  MoveL 7815 to (31.1, 13.35, -12.25) mm, rotated rx -180 ry 0 rz 90 deg; joints [74.527, -16.728, 82.289, 0, 24.439, 74.527]
  MoveL 7816 to (23.55, 13.35, -12.25) mm, rotated rx 180 ry 0 rz 90 deg; joints [74.46, -16.875, 82.836, 0, 24.039, 74.46]
  MoveL 7817 to (23.55, 15.07, -12.25) mm, rotated rx -180 ry 0 rz 90 deg; joints [74.516, -16.884, 82.871, 0, 24.013, 74.516]
  MoveL 7818 to (23.55, 15.07, -9.25) mm, rotated rx 180 ry 0 rz 90 deg; joints [74.516, -17.037, 82.973, 0, 24.064, 74.516]
  Establecer velocidad (1000.0 mm/s)
  MoveL 7819 to (23.55, 15.07, 10) mm, rotated rx 180 ry 0 rz 90 deg; joints [74.516, -18.015, 83.619, 0, 24.396, 74.516]
  Establecer velocidad (66.7 mm/s)
  MoveL 7820 to (-7.83, 65.77, 10) mm, rotated rx -180 ry 0 rz 90 deg; joints [75.899, -18.849, 86.805, 0, 22.044, 75.899]
  MoveL 7821 to (-7.83, 65.77, -9) mm, rotated rx 180 ry 0 rz 90 deg; joints [75.899, -17.87, 86.169, 0, 21.701, 75.899]
  MoveL 7822 to (-8.11, 64.28, -9.41) mm, rotated rx -180 ry 0 rz 90 deg; joints [75.847, -17.848, 86.149, 0, 21.699, 75.847]
  MoveL 7823 to (-7.99, 62.77, -9.81) mm, rotated rx -180 ry 0 rz 90 deg; joints [75.798, -17.818, 86.1, 0, 21.718, 75.798]
  MoveL 7824 to (-7.51, 61.33, -10.22) mm, rotated rx 180 ry 0 rz 90 deg; joints [75.754, -17.782, 86.027, 0, 21.756, 75.754]
  MoveL 7825 to (-6.7, 60.05, -10.62) mm, rotated rx -180 ry 0 rz 90 deg; joints [75.719, -17.742, 85.933, 0, 21.809, 75.719]
  MoveL 7826 to (-5.59, 59, -11.03) mm, rotated rx 180 ry 0 rz 90 deg; joints [75.693, -17.697, 85.823, 0, 21.874, 75.693]
  MoveL 7827 to (-4.27, 58.25, -11.44) mm, rotated rx -180 ry 0 rz 90 deg; joints [75.68, -17.649, 85.702, 0, 21.947, 75.68]
  MoveL 7828 to (-2.8, 57.85, -11.84) mm, rotated rx 180 ry 0 rz 90 deg; joints [75.679, -17.601, 85.578, 0, 22.023, 75.679]
  MoveL 7829 to (-1.29, 57.84, -12.25) mm, rotated rx 180 ry 0 rz 90 deg; joints [75.691, -17.553, 85.457, 0, 22.096, 75.691]
  MoveL 7830 to (6.58, 58.62, -12.25) mm, rotated rx 180 ry 0 rz 90 deg; joints [75.783, -17.416, 84.913, 0, 22.503, 75.783]
  MoveC 7831 to (18.86, 59.96, -12.25) mm, rotated rx 180 ry 0 rz 90 deg; joints [75.928, -17.197, 84.061, 0, 23.136, 75.928] to (31.1, 61.55, -12.25) mm, rotated rx -180 ry 0 rz 90 deg; joints [76.079, -16.973, 83.207, 0, 23.766, 76.079]
  MoveL 7832 to (31.1, 68.78, -12.25) mm, rotated rx 180 ry 0 rz 90 deg; joints [76.313, -17.007, 83.336, 0, 23.672, 76.313]
  MoveC 7833 to (8.53, 69.82, -12.25) mm, rotated rx -180 ry 0 rz 90 deg; joints [76.167, -17.432, 84.974, 0, 22.457, 76.167] to (-14.06, 70.54, -12.25) mm, rotated rx -180 ry 0 rz 90 deg; joints [76.005, -17.83, 86.579, 0, 21.251, 76.005]
  MoveC 7834 to (-16.19, 67.95, -12.25) mm, rotated rx -180 ry 0 rz 90 deg; joints [75.901, -17.855, 86.682, 0, 21.173, 75.901] to (-15.95, 64.6, -12.25) mm, rotated rx 180 ry 0 rz 90 deg; joints [75.792, -17.836, 86.606, 0, 21.231, 75.792]
  MoveL 7835 to (-7.11, 58.83, -12.25) mm, rotated rx 180 ry 0 rz 90 deg; joints [75.675, -17.66, 85.884, 0, 21.775, 75.675]
  MoveL 7836 to (-5.82, 57.95, -12.25) mm, rotated rx -180 ry 0 rz 90 deg; joints [75.657, -17.633, 85.778, 0, 21.855, 75.657]
  MoveC 7837 to (-5.45, 57.71, -12.25) mm, rotated rx 180 ry 0 rz 90 deg; joints [75.652, -17.626, 85.747, 0, 21.878, 75.652] to (-5.05, 57.51, -12.25) mm, rotated rx -180 ry 0 rz 90 deg; joints [75.649, -17.618, 85.716, 0, 21.902, 75.649]
  MoveC 7838 to (0.56, 58.01, -12.25) mm, rotated rx 180 ry 0 rz 90 deg; joints [75.713, -17.521, 85.329, 0, 22.192, 75.713] to (6.16, 58.57, -12.25) mm, rotated rx -180 ry 0 rz 90 deg; joints [75.778, -17.424, 84.943, 0, 22.481, 75.778]
  MoveC 7839 to (6.37, 58.59, -12.25) mm, rotated rx 180 ry 0 rz 90 deg; joints [75.78, -17.42, 84.928, 0, 22.492, 75.78] to (6.58, 58.62, -12.25) mm, rotated rx 180 ry 0 rz 90 deg; joints [75.783, -17.416, 84.913, 0, 22.503, 75.783]
  MoveL 7840 to (5.83, 66.13, -12.25) mm, rotated rx -180 ry 0 rz 90 deg; joints [76.023, -17.464, 85.101, 0, 22.363, 76.023]
  MoveL 7841 to (5.83, 66.13, -9.25) mm, rotated rx 180 ry 0 rz 90 deg; joints [76.023, -17.618, 85.203, 0, 22.415, 76.023]
  Establecer velocidad (1000.0 mm/s)
  MoveL 7842 to (5.83, 66.13, 10) mm, rotated rx 180 ry 0 rz 90 deg; joints [76.023, -18.605, 85.848, 0, 22.757, 76.023]
  Establecer velocidad (66.7 mm/s)
  MoveL 7843 to (-63.61, 35.65, 10) mm, rotated rx 180 ry 0 rz 90 deg; joints [74.395, -19.637, 90.091, 0, 19.546, 74.395]
  MoveL 7844 to (-63.61, 35.65, -9) mm, rotated rx 180 ry 0 rz 90 deg; joints [74.395, -18.644, 89.455, 0, 19.189, 74.395]
  MoveL 7845 to (-65.12, 35.84, -9.41) mm, rotated rx -180 ry 0 rz 90 deg; joints [74.387, -18.646, 89.546, 0, 19.1, 74.387]
  MoveL 7846 to (-66.63, 35.66, -9.81) mm, rotated rx -180 ry 0 rz 90 deg; joints [74.367, -18.646, 89.63, 0, 19.017, 74.367]
  MoveL 7847 to (-68.06, 35.14, -10.22) mm, rotated rx -180 ry 0 rz 90 deg; joints [74.336, -18.644, 89.702, 0, 18.942, 74.336]
  MoveL 7848 to (-69.34, 34.33, -10.62) mm, rotated rx 180 ry 0 rz 90 deg; joints [74.296, -18.639, 89.759, 0, 18.88, 74.296]
  MoveL 7849 to (-70.41, 33.25, -11.03) mm, rotated rx 180 ry 0 rz 90 deg; joints [74.249, -18.629, 89.796, 0, 18.832, 74.249]
  MoveL 7850 to (-71.21, 31.96, -11.44) mm, rotated rx 180 ry 0 rz 90 deg; joints [74.198, -18.614, 89.812, 0, 18.802, 74.198]
  MoveL 7851 to (-71.71, 30.53, -11.84) mm, rotated rx -180 ry 0 rz 90 deg; joints [74.144, -18.594, 89.804, 0, 18.79, 74.144]
  MoveL 7852 to (-71.85, 29.01, -12.25) mm, rotated rx -180 ry 0 rz 90 deg; joints [74.091, -18.568, 89.771, 0, 18.797, 74.091]
  MoveL 7853 to (-71.85, 4.26, -12.25) mm, rotated rx -180 ry 0 rz 90 deg; joints [73.256, -18.461, 89.286, 0, 19.175, 73.256]
  MoveL 7854 to (-71.84, 3.32, -12.25) mm, rotated rx -180 ry 0 rz 90 deg; joints [73.224, -18.456, 89.266, 0, 19.19, 73.224]
  MoveC 7855 to (-70.64, 1.17, -12.25) mm, rotated rx -180 ry 0 rz 90 deg; joints [73.164, -18.429, 89.142, 0, 19.287, 73.164] to (-68.23, 0.7, -12.25) mm, rotated rx -180 ry 0 rz 90 deg; joints [73.173, -18.39, 88.971, 0, 19.419, 73.173]
  MoveC 7856 to (-46.18, 5.94, -12.25) mm, rotated rx -180 ry 0 rz 90 deg; joints [73.567, -18.07, 87.584, 0, 20.486, 73.567] to (-24.17, 11.28, -12.25) mm, rotated rx 180 ry 0 rz 90 deg; joints [73.955, -17.731, 86.174, 0, 21.557, 73.955]
  MoveC 7857 to (-22.94, 12.16, -12.25) mm, rotated rx 180 ry 0 rz 90 deg; joints [73.996, -17.715, 86.107, 0, 21.607, 73.996] to (-22.27, 13.51, -12.25) mm, rotated rx 180 ry 0 rz 90 deg; joints [74.046, -17.71, 86.087, 0, 21.622, 74.046]
  MoveC 7858 to (-22.16, 14.34, -12.25) mm, rotated rx -180 ry 0 rz 90 deg; joints [74.075, -17.712, 86.096, 0, 21.616, 74.075] to (-22.32, 15.16, -12.25) mm, rotated rx -180 ry 0 rz 90 deg; joints [74.1, -17.719, 86.123, 0, 21.595, 74.1]
  MoveL 7859 to (-22.48, 15.64, -12.25) mm, rotated rx -180 ry 0 rz 90 deg; joints [74.114, -17.724, 86.144, 0, 21.58, 74.114]
  MoveL 7860 to (-27.68, 30.34, -12.25) mm, rotated rx 180 ry 0 rz 90 deg; joints [74.551, -17.881, 86.791, 0, 21.09, 74.551]
  MoveC 7861 to (-28.18, 31.24, -12.25) mm, rotated rx -180 ry 0 rz 90 deg; joints [74.577, -17.894, 86.843, 0, 21.051, 74.577] to (-28.94, 31.94, -12.25) mm, rotated rx 180 ry 0 rz 90 deg; joints [74.593, -17.91, 86.909, 0, 21.001, 74.593]
  MoveC 7862 to (-48.2, 44.55, -12.25) mm, rotated rx -180 ry 0 rz 90 deg; joints [74.838, -18.275, 88.466, 0, 19.809, 74.838] to (-67.5, 57.09, -12.25) mm, rotated rx -180 ry 0 rz 90 deg; joints [75.088, -18.618, 89.998, 0, 18.62, 75.088]
  MoveC 7863 to (-67.85, 57.26, -12.25) mm, rotated rx 180 ry 0 rz 90 deg; joints [75.09, -18.624, 90.024, 0, 18.599, 75.09] to (-68.23, 57.34, -12.25) mm, rotated rx 180 ry 0 rz 90 deg; joints [75.089, -18.629, 90.051, 0, 18.578, 75.089]
  MoveC 7864 to (-70.13, 56.97, -12.25) mm, rotated rx -180 ry 0 rz 90 deg; joints [75.059, -18.655, 90.172, 0, 18.484, 75.059] to (-71.56, 55.68, -12.25) mm, rotated rx -180 ry 0 rz 90 deg; joints [75.002, -18.671, 90.245, 0, 18.427, 75.002]
  MoveC 7865 to (-71.78, 55.22, -12.25) mm, rotated rx -180 ry 0 rz 90 deg; joints [74.985, -18.672, 90.251, 0, 18.422, 74.985] to (-71.85, 54.71, -12.25) mm, rotated rx 180 ry 0 rz 90 deg; joints [74.967, -18.672, 90.247, 0, 18.425, 74.967]
  MoveL 7866 to (-71.85, 29.01, -12.25) mm, rotated rx -180 ry 0 rz 90 deg; joints [74.091, -18.568, 89.771, 0, 18.797, 74.091]
  MoveL 7867 to (-64.3, 29.01, -12.25) mm, rotated rx 180 ry 0 rz 90 deg; joints [74.164, -18.456, 89.264, 0, 19.192, 74.164]
  MoveL 7868 to (-64.3, 29.01, -9.25) mm, rotated rx 180 ry 0 rz 90 deg; joints [74.164, -18.613, 89.367, 0, 19.246, 74.164]
  Establecer velocidad (1000.0 mm/s)
  MoveL 7869 to (-64.3, 29.01, 10) mm, rotated rx 180 ry 0 rz 90 deg; joints [74.164, -19.619, 90.012, 0, 19.607, 74.164]
  Establecer velocidad (66.7 mm/s)
  MoveL 7870 to (-63.45, 35.65, 10) mm, rotated rx -180 ry 0 rz 90 deg; joints [74.397, -19.635, 90.08, 0, 19.555, 74.397]
  MoveL 7871 to (-63.45, 35.65, -9.25) mm, rotated rx 180 ry 0 rz 90 deg; joints [74.397, -18.628, 89.435, 0, 19.193, 74.397]
  MoveL 7872 to (-64.95, 35.84, -9.66) mm, rotated rx -180 ry 0 rz 90 deg; joints [74.389, -18.63, 89.526, 0, 19.104, 74.389]
  MoveL 7873 to (-66.46, 35.66, -10.06) mm, rotated rx 180 ry 0 rz 90 deg; joints [74.368, -18.631, 89.61, 0, 19.021, 74.368]
  MoveL 7874 to (-67.89, 35.14, -10.47) mm, rotated rx -180 ry 0 rz 90 deg; joints [74.337, -18.629, 89.682, 0, 18.946, 74.337]
  MoveL 7875 to (-69.17, 34.33, -10.87) mm, rotated rx -180 ry 0 rz 90 deg; joints [74.297, -18.623, 89.739, 0, 18.884, 74.297]
  MoveL 7876 to (-70.24, 33.25, -11.28) mm, rotated rx 180 ry 0 rz 90 deg; joints [74.251, -18.613, 89.777, 0, 18.836, 74.251]
  MoveL 7877 to (-71.05, 31.96, -11.69) mm, rotated rx -180 ry 0 rz 90 deg; joints [74.199, -18.598, 89.792, 0, 18.806, 74.199]
  MoveL 7878 to (-71.55, 30.53, -12.09) mm, rotated rx 180 ry 0 rz 90 deg; joints [74.146, -18.578, 89.785, 0, 18.794, 74.146]
  MoveL 7879 to (-71.69, 29.01, -12.5) mm, rotated rx 180 ry 0 rz 90 deg; joints [74.093, -18.553, 89.751, 0, 18.801, 74.093]
  MoveL 7880 to (-71.69, 4.26, -12.5) mm, rotated rx 180 ry 0 rz 90 deg; joints [73.257, -18.445, 89.266, 0, 19.179, 73.257]
  MoveL 7881 to (-71.67, 3.32, -12.5) mm, rotated rx -180 ry 0 rz 90 deg; joints [73.226, -18.441, 89.246, 0, 19.195, 73.226]
  MoveC 7882 to (-70.48, 1.34, -12.5) mm, rotated rx -180 ry 0 rz 90 deg; joints [73.171, -18.414, 89.126, 0, 19.288, 73.171] to (-68.23, 0.85, -12.5) mm, rotated rx 180 ry 0 rz 90 deg; joints [73.178, -18.378, 88.965, 0, 19.413, 73.178]
  MoveC 7883 to (-46.66, 5.98, -12.5) mm, rotated rx 180 ry 0 rz 90 deg; joints [73.564, -18.065, 87.609, 0, 20.457, 73.564] to (-25.11, 11.2, -12.5) mm, rotated rx 180 ry 0 rz 90 deg; joints [73.944, -17.734, 86.23, 0, 21.504, 73.944]
  MoveL 7884 to (-24.61, 11.33, -12.5) mm, rotated rx -180 ry 0 rz 90 deg; joints [73.953, -17.726, 86.198, 0, 21.528, 73.953]
  MoveC 7885 to (-23.47, 11.94, -12.5) mm, rotated rx 180 ry 0 rz 90 deg; joints [73.983, -17.71, 86.13, 0, 21.579, 73.983] to (-22.73, 13, -12.5) mm, rotated rx 180 ry 0 rz 90 deg; joints [74.025, -17.702, 86.101, 0, 21.602, 74.025]
  MoveL 7886 to (-22.44, 13.74, -12.5) mm, rotated rx -180 ry 0 rz 90 deg; joints [74.052, -17.701, 86.095, 0, 21.606, 74.052]
  MoveL 7887 to (-22.37, 14.21, -12.5) mm, rotated rx 180 ry 0 rz 90 deg; joints [74.069, -17.702, 86.1, 0, 21.602, 74.069]
  MoveL 7888 to (-22.38, 14.69, -12.5) mm, rotated rx -180 ry 0 rz 90 deg; joints [74.084, -17.704, 86.11, 0, 21.595, 74.084]
  MoveL 7889 to (-22.49, 15.16, -12.5) mm, rotated rx -180 ry 0 rz 90 deg; joints [74.099, -17.709, 86.127, 0, 21.582, 74.099]
  MoveL 7890 to (-22.65, 15.64, -12.5) mm, rotated rx 180 ry 0 rz 90 deg; joints [74.113, -17.714, 86.147, 0, 21.567, 74.113]
  MoveL 7891 to (-27.81, 30.22, -12.5) mm, rotated rx 180 ry 0 rz 90 deg; joints [74.546, -17.87, 86.789, 0, 21.081, 74.546]
  MoveC 7892 to (-28.31, 31.13, -12.5) mm, rotated rx -180 ry 0 rz 90 deg; joints [74.572, -17.882, 86.841, 0, 21.042, 74.572] to (-29.07, 31.83, -12.5) mm, rotated rx -180 ry 0 rz 90 deg; joints [74.588, -17.898, 86.907, 0, 20.991, 74.588]
  MoveC 7893 to (-48.17, 44.36, -12.5) mm, rotated rx 180 ry 0 rz 90 deg; joints [74.832, -18.261, 88.452, 0, 19.809, 74.832] to (-67.31, 56.8, -12.5) mm, rotated rx -180 ry 0 rz 90 deg; joints [75.08, -18.601, 89.971, 0, 18.629, 75.08]
  MoveC 7894 to (-67.75, 57.01, -12.5) mm, rotated rx -180 ry 0 rz 90 deg; joints [75.083, -18.608, 90.005, 0, 18.603, 75.083] to (-68.23, 57.1, -12.5) mm, rotated rx 180 ry 0 rz 90 deg; joints [75.081, -18.615, 90.038, 0, 18.577, 75.081]
  MoveC 7895 to (-70.04, 56.69, -12.5) mm, rotated rx 180 ry 0 rz 90 deg; joints [75.051, -18.64, 90.152, 0, 18.488, 75.051] to (-71.41, 55.44, -12.5) mm, rotated rx -180 ry 0 rz 90 deg; joints [74.996, -18.655, 90.221, 0, 18.434, 74.996]
  MoveC 7896 to (-71.62, 54.99, -12.5) mm, rotated rx -180 ry 0 rz 90 deg; joints [74.978, -18.656, 90.227, 0, 18.429, 74.978] to (-71.69, 54.49, -12.5) mm, rotated rx -180 ry 0 rz 90 deg; joints [74.961, -18.655, 90.223, 0, 18.432, 74.961]
  MoveL 7897 to (-71.69, 29.01, -12.5) mm, rotated rx 180 ry 0 rz 90 deg; joints [74.093, -18.553, 89.751, 0, 18.801, 74.093]
  MoveL 7898 to (-64.14, 29.01, -12.5) mm, rotated rx -180 ry 0 rz 90 deg; joints [74.166, -18.441, 89.245, 0, 19.196, 74.166]
  MoveL 7899 to (-64.14, 29.01, -9.5) mm, rotated rx -180 ry 0 rz 90 deg; joints [74.166, -18.598, 89.347, 0, 19.25, 74.166]
  Establecer velocidad (1000.0 mm/s)
  MoveL 7900 to (-64.14, 29.01, 10) mm, rotated rx 180 ry 0 rz 90 deg; joints [74.166, -19.617, 90.001, 0, 19.616, 74.166]
  Establecer velocidad (66.7 mm/s)
  MoveL 7901 to (-6.74, 60.15, 10) mm, rotated rx -180 ry 0 rz 90 deg; joints [75.722, -18.804, 86.629, 0, 22.176, 75.722]
  MoveL 7902 to (-6.74, 60.15, -9.25) mm, rotated rx -180 ry 0 rz 90 deg; joints [75.722, -17.814, 85.984, 0, 21.829, 75.722]
  MoveL 7903 to (-5.66, 59.08, -9.66) mm, rotated rx -180 ry 0 rz 90 deg; joints [75.696, -17.769, 85.876, 0, 21.893, 75.696]
  MoveL 7904 to (-4.34, 58.34, -10.06) mm, rotated rx -180 ry 0 rz 90 deg; joints [75.682, -17.722, 85.755, 0, 21.966, 75.682]
  MoveL 7905 to (-2.87, 57.95, -10.47) mm, rotated rx 180 ry 0 rz 90 deg; joints [75.682, -17.673, 85.631, 0, 22.042, 75.682]
  MoveL 7906 to (-1.35, 57.93, -10.87) mm, rotated rx -180 ry 0 rz 90 deg; joints [75.694, -17.625, 85.51, 0, 22.116, 75.694]
  MoveL 7907 to (0.13, 58.3, -11.28) mm, rotated rx -180 ry 0 rz 90 deg; joints [75.718, -17.58, 85.398, 0, 22.182, 75.718]
  MoveL 7908 to (1.47, 59.02, -11.69) mm, rotated rx 180 ry 0 rz 90 deg; joints [75.753, -17.539, 85.302, 0, 22.236, 75.753]
  MoveL 7909 to (2.59, 60.05, -12.09) mm, rotated rx 180 ry 0 rz 90 deg; joints [75.797, -17.502, 85.228, 0, 22.274, 75.797]
  MoveL 7910 to (3.39, 61.34, -12.5) mm, rotated rx 180 ry 0 rz 90 deg; joints [75.846, -17.473, 85.18, 0, 22.293, 75.846]
  MoveL 7911 to (7.41, 69.66, -12.5) mm, rotated rx 180 ry 0 rz 90 deg; joints [76.152, -17.438, 85.042, 0, 22.396, 76.152]
  MoveC 7912 to (-3.01, 70.04, -12.5) mm, rotated rx -180 ry 0 rz 90 deg; joints [76.08, -17.625, 85.786, 0, 21.838, 76.08] to (-13.44, 70.34, -12.5) mm, rotated rx 180 ry 0 rz 90 deg; joints [76.004, -17.806, 86.523, 0, 21.283, 76.004]
  MoveC 7913 to (-15.54, 67.78, -12.5) mm, rotated rx 180 ry 0 rz 90 deg; joints [75.901, -17.83, 86.625, 0, 21.205, 75.901] to (-15.31, 64.47, -12.5) mm, rotated rx 180 ry 0 rz 90 deg; joints [75.793, -17.812, 86.551, 0, 21.262, 75.793]
  MoveL 7914 to (-7.11, 59.11, -12.5) mm, rotated rx 180 ry 0 rz 90 deg; joints [75.685, -17.648, 85.881, 0, 21.767, 75.685]
  MoveL 7915 to (-5.19, 57.81, -12.5) mm, rotated rx 180 ry 0 rz 90 deg; joints [75.657, -17.609, 85.723, 0, 21.886, 75.657]
  MoveL 7916 to (-4.86, 57.65, -12.5) mm, rotated rx 180 ry 0 rz 90 deg; joints [75.655, -17.602, 85.696, 0, 21.906, 75.655]
  MoveC 7917 to (11.72, 59.29, -12.5) mm, rotated rx -180 ry 0 rz 90 deg; joints [75.847, -17.313, 84.552, 0, 22.761, 75.847] to (28.24, 61.34, -12.5) mm, rotated rx -180 ry 0 rz 90 deg; joints [76.049, -17.014, 83.401, 0, 23.613, 76.049]
  MoveL 7918 to (28.24, 68.7, -12.5) mm, rotated rx -180 ry 0 rz 90 deg; joints [76.288, -17.049, 83.532, 0, 23.516, 76.288]
  MoveC 7919 to (17.83, 69.22, -12.5) mm, rotated rx 180 ry 0 rz 90 deg; joints [76.222, -17.246, 84.291, 0, 22.955, 76.222] to (7.41, 69.66, -12.5) mm, rotated rx 180 ry 0 rz 90 deg; joints [76.152, -17.438, 85.042, 0, 22.396, 76.152]
  MoveL 7920 to (7.11, 62.12, -12.5) mm, rotated rx 180 ry 0 rz 90 deg; joints [75.902, -17.41, 84.93, 0, 22.48, 75.902]
  MoveL 7921 to (7.11, 62.12, -9.5) mm, rotated rx -180 ry 0 rz 90 deg; joints [75.902, -17.564, 85.032, 0, 22.531, 75.902]
  Establecer velocidad (1000.0 mm/s)
  MoveL 7922 to (7.11, 62.12, 10) mm, rotated rx 180 ry 0 rz 90 deg; joints [75.902, -18.563, 85.686, 0, 22.878, 75.902]
  Establecer velocidad (66.7 mm/s)
  MoveL 7923 to (15.22, 14.3, 10) mm, rotated rx -180 ry 0 rz 90 deg; joints [74.416, -18.173, 84.203, 0, 23.97, 74.416]
  MoveL 7924 to (15.22, 14.3, -9.25) mm, rotated rx -180 ry 0 rz 90 deg; joints [74.416, -17.192, 83.557, 0, 23.635, 74.416]
  MoveL 7925 to (15.95, 12.97, -9.66) mm, rotated rx -180 ry 0 rz 90 deg; joints [74.38, -17.15, 83.464, 0, 23.686, 74.38]
  MoveL 7926 to (16.98, 11.85, -10.06) mm, rotated rx 180 ry 0 rz 90 deg; joints [74.353, -17.104, 83.354, 0, 23.75, 74.353]
  MoveL 7927 to (18.23, 10.99, -10.47) mm, rotated rx -180 ry 0 rz 90 deg; joints [74.337, -17.055, 83.233, 0, 23.822, 74.337]
  MoveL 7928 to (19.65, 10.43, -10.87) mm, rotated rx -180 ry 0 rz 90 deg; joints [74.332, -17.004, 83.106, 0, 23.898, 74.332]
  MoveL 7929 to (21.15, 10.19, -11.28) mm, rotated rx 180 ry 0 rz 90 deg; joints [74.338, -16.953, 82.979, 0, 23.974, 74.338]
  MoveL 7930 to (22.66, 10.29, -11.69) mm, rotated rx 180 ry 0 rz 90 deg; joints [74.355, -16.904, 82.858, 0, 24.046, 74.355]
  MoveL 7931 to (24.12, 10.73, -12.09) mm, rotated rx -180 ry 0 rz 90 deg; joints [74.382, -16.858, 82.748, 0, 24.11, 74.382]
  MoveL 7932 to (25.43, 11.5, -12.5) mm, rotated rx -180 ry 0 rz 90 deg; joints [74.418, -16.816, 82.655, 0, 24.161, 74.418]
  MoveL 7933 to (28.24, 13.53, -12.5) mm, rotated rx 180 ry 0 rz 90 deg; joints [74.508, -16.772, 82.492, 0, 24.28, 74.508]
  MoveL 7934 to (28.24, 24.45, -12.5) mm, rotated rx 180 ry 0 rz 90 deg; joints [74.858, -16.83, 82.708, 0, 24.122, 74.858]
  MoveL 7935 to (27.01, 24.48, -12.5) mm, rotated rx -180 ry 0 rz 90 deg; joints [74.848, -16.854, 82.799, 0, 24.056, 74.848]
  MoveL 7936 to (16.58, 24.56, -12.5) mm, rotated rx 180 ry 0 rz 90 deg; joints [74.76, -17.054, 83.551, 0, 23.502, 74.76]
  MoveL 7937 to (15.64, 24.53, -12.5) mm, rotated rx 180 ry 0 rz 90 deg; joints [74.75, -17.071, 83.619, 0, 23.452, 74.75]
  MoveC 7938 to (13.67, 23.69, -12.5) mm, rotated rx -180 ry 0 rz 90 deg; joints [74.706, -17.104, 83.743, 0, 23.361, 74.706] to (12.68, 21.8, -12.5) mm, rotated rx 180 ry 0 rz 90 deg; joints [74.636, -17.113, 83.777, 0, 23.336, 74.636]
  MoveC 7939 to (12.67, 21.32, -12.5) mm, rotated rx -180 ry 0 rz 90 deg; joints [74.62, -17.111, 83.768, 0, 23.342, 74.62] to (12.77, 20.85, -12.5) mm, rotated rx -180 ry 0 rz 90 deg; joints [74.606, -17.106, 83.752, 0, 23.354, 74.606]
  MoveL 7940 to (16.01, 12.15, -12.5) mm, rotated rx 180 ry 0 rz 90 deg; joints [74.354, -17, 83.347, 0, 23.653, 74.354]
  MoveC 7941 to (16.44, 11.37, -12.5) mm, rotated rx -180 ry 0 rz 90 deg; joints [74.333, -16.988, 83.3, 0, 23.687, 74.333] to (17.07, 10.75, -12.5) mm, rotated rx 180 ry 0 rz 90 deg; joints [74.319, -16.972, 83.242, 0, 23.73, 74.319]
  MoveL 7942 to (27.26, 3.32, -12.5) mm, rotated rx -180 ry 0 rz 90 deg; joints [74.173, -16.735, 82.355, 0, 24.38, 74.173]
  MoveL 7943 to (28.24, 2.61, -12.5) mm, rotated rx 180 ry 0 rz 90 deg; joints [74.159, -16.712, 82.269, 0, 24.443, 74.159]
  MoveL 7944 to (28.24, 13.53, -12.5) mm, rotated rx 180 ry 0 rz 90 deg; joints [74.508, -16.772, 82.492, 0, 24.28, 74.508]
  MoveL 7945 to (20.7, 13.53, -12.5) mm, rotated rx -180 ry 0 rz 90 deg; joints [74.441, -16.918, 83.037, 0, 23.88, 74.441]
  MoveL 7946 to (20.7, 13.53, -9.5) mm, rotated rx -180 ry 0 rz 90 deg; joints [74.441, -17.071, 83.14, 0, 23.931, 74.441]
  Establecer velocidad (1000.0 mm/s)
  MoveL 7947 to (20.7, 13.53, 10) mm, rotated rx 180 ry 0 rz 90 deg; joints [74.441, -18.063, 83.794, 0, 24.268, 74.441]
  Establecer velocidad (66.7 mm/s)
  MoveL 7948 to (14.69, -46.1, 10) mm, rotated rx -180 ry 0 rz 90 deg; joints [72.484, -17.833, 82.952, 0, 24.881, 72.484]
  MoveL 7949 to (14.69, -46.1, -9.25) mm, rotated rx 180 ry 0 rz 90 deg; joints [72.484, -16.857, 82.305, 0, 24.551, 72.484]
  MoveL 7950 to (13.29, -45.53, -9.66) mm, rotated rx 180 ry 0 rz 90 deg; joints [72.488, -16.867, 82.405, 0, 24.462, 72.488]
  MoveL 7951 to (11.79, -45.31, -10.06) mm, rotated rx -180 ry 0 rz 90 deg; joints [72.48, -16.877, 82.505, 0, 24.372, 72.48]
  MoveL 7952 to (10.27, -45.43, -10.47) mm, rotated rx 180 ry 0 rz 90 deg; joints [72.461, -16.885, 82.597, 0, 24.288, 72.461]
  MoveL 7953 to (8.82, -45.87, -10.87) mm, rotated rx 180 ry 0 rz 90 deg; joints [72.432, -16.889, 82.677, 0, 24.213, 72.432]
  MoveL 7954 to (7.5, -46.63, -11.28) mm, rotated rx -180 ry 0 rz 90 deg; joints [72.395, -16.889, 82.74, 0, 24.15, 72.395]
  MoveL 7955 to (6.39, -47.67, -11.69) mm, rotated rx 180 ry 0 rz 90 deg; joints [72.351, -16.884, 82.782, 0, 24.102, 72.351]
  MoveL 7956 to (5.53, -48.92, -12.09) mm, rotated rx -180 ry 0 rz 90 deg; joints [72.303, -16.872, 82.801, 0, 24.071, 72.303]
  MoveL 7957 to (5, -50.34, -12.5) mm, rotated rx -180 ry 0 rz 90 deg; joints [72.252, -16.853, 82.793, 0, 24.06, 72.252]
  MoveL 7958 to (0.65, -66.33, -12.5) mm, rotated rx 180 ry 0 rz 90 deg; joints [71.701, -16.836, 82.732, 0, 24.104, 71.701]
  MoveL 7959 to (0.54, -66.81, -12.5) mm, rotated rx 180 ry 0 rz 90 deg; joints [71.685, -16.835, 82.728, 0, 24.107, 71.685]
  MoveC 7960 to (1.32, -68.93, -12.5) mm, rotated rx -180 ry 0 rz 90 deg; joints [71.627, -16.807, 82.623, 0, 24.185, 71.627] to (3.32, -69.98, -12.5) mm, rotated rx -180 ry 0 rz 90 deg; joints [71.614, -16.762, 82.455, 0, 24.307, 71.614]
  MoveL 7961 to (4.26, -69.98, -12.5) mm, rotated rx 180 ry 0 rz 90 deg; joints [71.624, -16.744, 82.387, 0, 24.356, 71.624]
  MoveC 7962 to (16.26, -69.52, -12.5) mm, rotated rx -180 ry 0 rz 90 deg; joints [71.763, -16.512, 81.536, 0, 24.976, 71.763] to (28.24, -68.93, -12.5) mm, rotated rx 180 ry 0 rz 90 deg; joints [71.905, -16.275, 80.68, 0, 25.595, 71.905]
  MoveL 7963 to (28.24, -47.07, -12.5) mm, rotated rx -180 ry 0 rz 90 deg; joints [72.588, -16.417, 81.19, 0, 25.226, 72.588]
  MoveL 7964 to (27.35, -45.96, -12.5) mm, rotated rx 180 ry 0 rz 90 deg; joints [72.614, -16.442, 81.28, 0, 25.161, 72.614]
  MoveL 7965 to (22.76, -40.34, -12.5) mm, rotated rx 180 ry 0 rz 90 deg; joints [72.745, -16.568, 81.741, 0, 24.827, 72.745]
  MoveC 7966 to (22.34, -39.87, -12.5) mm, rotated rx -180 ry 0 rz 90 deg; joints [72.756, -16.579, 81.782, 0, 24.797, 72.756] to (21.88, -39.45, -12.5) mm, rotated rx -180 ry 0 rz 90 deg; joints [72.765, -16.591, 81.825, 0, 24.766, 72.765]
  MoveL 7967 to (14.21, -33.04, -12.5) mm, rotated rx 180 ry 0 rz 90 deg; joints [72.893, -16.78, 82.521, 0, 24.258, 72.893]
  MoveC 7968 to (11.72, -32.6, -12.5) mm, rotated rx 180 ry 0 rz 90 deg; joints [72.882, -16.831, 82.711, 0, 24.12, 72.882] to (9.54, -33.9, -12.5) mm, rotated rx 180 ry 0 rz 90 deg; joints [72.82, -16.865, 82.838, 0, 24.027, 72.82]
  MoveL 7969 to (9.48, -34.03, -12.5) mm, rotated rx 180 ry 0 rz 90 deg; joints [72.815, -16.865, 82.839, 0, 24.026, 72.815]
  MoveL 7970 to (6.71, -44.07, -12.5) mm, rotated rx -180 ry 0 rz 90 deg; joints [72.469, -16.858, 82.813, 0, 24.045, 72.469]
  MoveL 7971 to (5, -50.34, -12.5) mm, rotated rx -180 ry 0 rz 90 deg; joints [72.252, -16.853, 82.793, 0, 24.06, 72.252]
  MoveL 7972 to (12.28, -52.33, -12.5) mm, rotated rx 180 ry 0 rz 90 deg; joints [72.263, -16.7, 82.225, 0, 24.475, 72.263]
  MoveL 7973 to (12.28, -52.33, -9.5) mm, rotated rx 180 ry 0 rz 90 deg; joints [72.263, -16.852, 82.328, 0, 24.525, 72.263]
  Establecer velocidad (1000.0 mm/s)
  MoveL 7974 to (12.28, -52.33, 10) mm, rotated rx 180 ry 0 rz 90 deg; joints [72.263, -17.842, 82.983, 0, 24.859, 72.263]
  Establecer velocidad (66.7 mm/s)
  MoveL 7975 to (-38.53, -51.97, 10) mm, rotated rx -180 ry 0 rz 90 deg; joints [71.747, -18.788, 86.565, 0, 22.224, 71.747]
  MoveL 7976 to (-38.53, -51.97, -9.25) mm, rotated rx 180 ry 0 rz 90 deg; joints [71.747, -17.798, 85.92, 0, 21.878, 71.747]
  MoveL 7977 to (-37.12, -52.52, -9.66) mm, rotated rx 180 ry 0 rz 90 deg; joints [71.744, -17.749, 85.796, 0, 21.953, 71.744]
  MoveL 7978 to (-35.61, -52.72, -10.06) mm, rotated rx -180 ry 0 rz 90 deg; joints [71.754, -17.701, 85.674, 0, 22.027, 71.754]
  MoveL 7979 to (-34.1, -52.58, -10.47) mm, rotated rx -180 ry 0 rz 90 deg; joints [71.774, -17.655, 85.559, 0, 22.096, 71.774]
  MoveL 7980 to (-32.65, -52.11, -10.87) mm, rotated rx 180 ry 0 rz 90 deg; joints [71.805, -17.612, 85.456, 0, 22.156, 71.805]
  MoveL 7981 to (-31.35, -51.33, -11.28) mm, rotated rx 180 ry 0 rz 90 deg; joints [71.844, -17.573, 85.369, 0, 22.204, 71.844]
  MoveL 7982 to (-30.25, -50.28, -11.69) mm, rotated rx -180 ry 0 rz 90 deg; joints [71.889, -17.539, 85.303, 0, 22.236, 71.889]
  MoveL 7983 to (-29.41, -49.02, -12.09) mm, rotated rx -180 ry 0 rz 90 deg; joints [71.939, -17.51, 85.259, 0, 22.251, 71.939]
  MoveL 7984 to (-28.9, -47.59, -12.5) mm, rotated rx -180 ry 0 rz 90 deg; joints [71.991, -17.489, 85.242, 0, 22.246, 71.991]
  MoveL 7985 to (-23.6, -27.01, -12.5) mm, rotated rx -180 ry 0 rz 90 deg; joints [72.711, -17.511, 85.33, 0, 22.181, 72.711]
  MoveL 7986 to (-23.49, -26.54, -12.5) mm, rotated rx -180 ry 0 rz 90 deg; joints [72.727, -17.511, 85.332, 0, 22.179, 72.727]
  MoveC 7987 to (-23.63, -25.39, -12.5) mm, rotated rx 180 ry 0 rz 90 deg; joints [72.763, -17.52, 85.366, 0, 22.153, 72.763] to (-24.17, -24.36, -12.5) mm, rotated rx -180 ry 0 rz 90 deg; joints [72.791, -17.535, 85.426, 0, 22.109, 72.791]
  MoveC 7988 to (-25.19, -23.36, -12.5) mm, rotated rx -180 ry 0 rz 90 deg; joints [72.813, -17.558, 85.519, 0, 22.039, 72.813] to (-26.54, -22.86, -12.5) mm, rotated rx 180 ry 0 rz 90 deg; joints [72.816, -17.584, 85.623, 0, 21.961, 72.816]
  MoveL 7989 to (-27.01, -22.92, -12.5) mm, rotated rx 180 ry 0 rz 90 deg; joints [72.809, -17.592, 85.654, 0, 21.937, 72.809]
  MoveL 7990 to (-43.39, -26.21, -12.5) mm, rotated rx -180 ry 0 rz 90 deg; joints [72.535, -17.852, 86.714, 0, 21.138, 72.535]
  MoveC 7991 to (-56.45, -28.85, -12.5) mm, rotated rx 180 ry 0 rz 90 deg; joints [72.312, -18.051, 87.548, 0, 20.503, 72.312] to (-69.51, -31.54, -12.5) mm, rotated rx 180 ry 0 rz 90 deg; joints [72.085, -18.243, 88.371, 0, 19.872, 72.085]
  MoveC 7992 to (-70.66, -32.08, -12.5) mm, rotated rx -180 ry 0 rz 90 deg; joints [72.055, -18.258, 88.436, 0, 19.821, 72.055] to (-71.43, -33.09, -12.5) mm, rotated rx 180 ry 0 rz 90 deg; joints [72.013, -18.264, 88.466, 0, 19.798, 72.013]
  MoveC 7993 to (-71.62, -33.69, -12.5) mm, rotated rx -180 ry 0 rz 90 deg; joints [71.991, -18.264, 88.466, 0, 19.799, 71.991] to (-71.69, -34.31, -12.5) mm, rotated rx 180 ry 0 rz 90 deg; joints [71.97, -18.262, 88.457, 0, 19.806, 71.97]
  MoveL 7994 to (-71.69, -67.76, -12.5) mm, rotated rx 180 ry 0 rz 90 deg; joints [70.868, -18.087, 87.702, 0, 20.385, 70.868]
  MoveL 7995 to (-71.68, -68.54, -12.5) mm, rotated rx 180 ry 0 rz 90 deg; joints [70.842, -18.083, 87.683, 0, 20.4, 70.842]
  MoveC 7996 to (-70.83, -70.55, -12.5) mm, rotated rx 180 ry 0 rz 90 deg; joints [70.787, -18.058, 87.579, 0, 20.479, 70.787] to (-68.81, -71.36, -12.5) mm, rotated rx -180 ry 0 rz 90 deg; joints [70.783, -18.022, 87.424, 0, 20.598, 70.783]
  MoveC 7997 to (-52.95, -71.11, -12.5) mm, rotated rx 180 ry 0 rz 90 deg; joints [70.97, -17.765, 86.355, 0, 21.409, 70.97] to (-37.1, -70.81, -12.5) mm, rotated rx 180 ry 0 rz 90 deg; joints [71.155, -17.497, 85.274, 0, 22.222, 71.155]
  MoveC 7998 to (-36.96, -70.81, -12.5) mm, rotated rx 180 ry 0 rz 90 deg; joints [71.157, -17.494, 85.265, 0, 22.23, 71.157] to (-36.81, -70.79, -12.5) mm, rotated rx -180 ry 0 rz 90 deg; joints [71.159, -17.492, 85.255, 0, 22.237, 71.159]
  MoveC 7999 to (-35.24, -70.11, -12.5) mm, rotated rx 180 ry 0 rz 90 deg; joints [71.198, -17.468, 85.162, 0, 22.306, 71.198] to (-34.33, -68.64, -12.5) mm, rotated rx 180 ry 0 rz 90 deg; joints [71.255, -17.461, 85.134, 0, 22.328, 71.255]
  MoveL 8000 to (-32.86, -63.02, -12.5) mm, rotated rx 180 ry 0 rz 90 deg; joints [71.451, -17.469, 85.164, 0, 22.305, 71.451]
  MoveL 8001 to (-28.9, -47.59, -12.5) mm, rotated rx -180 ry 0 rz 90 deg; joints [71.991, -17.489, 85.242, 0, 22.246, 71.991]
  MoveL 8002 to (-36.21, -45.71, -12.5) mm, rotated rx 180 ry 0 rz 90 deg; joints [71.974, -17.626, 85.791, 0, 21.835, 71.974]
  MoveL 8003 to (-36.21, -45.71, -9.5) mm, rotated rx 180 ry 0 rz 90 deg; joints [71.974, -17.78, 85.893, 0, 21.887, 71.974]
  Establecer velocidad (1000.0 mm/s)
  MoveL 8004 to (-36.21, -45.71, 10) mm, rotated rx -180 ry 0 rz 90 deg; joints [71.974, -18.784, 86.546, 0, 22.237, 71.974]
  Establecer velocidad (66.7 mm/s)
  MoveL 8005 to (-38.68, -51.94, 10) mm, rotated rx -180 ry 0 rz 90 deg; joints [71.747, -18.791, 86.576, 0, 22.215, 71.747]
  MoveL 8006 to (-38.68, -51.94, -9.5) mm, rotated rx -180 ry 0 rz 90 deg; joints [71.747, -17.788, 85.923, 0, 21.865, 71.747]
  MoveL 8007 to (-37.27, -52.49, -9.91) mm, rotated rx 180 ry 0 rz 90 deg; joints [71.744, -17.739, 85.799, 0, 21.94, 71.744]
  MoveL 8008 to (-35.77, -52.68, -10.31) mm, rotated rx 180 ry 0 rz 90 deg; joints [71.753, -17.691, 85.677, 0, 22.014, 71.753]
  MoveL 8009 to (-34.25, -52.54, -10.72) mm, rotated rx 180 ry 0 rz 90 deg; joints [71.774, -17.645, 85.562, 0, 22.083, 71.774]
  MoveL 8010 to (-32.81, -52.08, -11.13) mm, rotated rx -180 ry 0 rz 90 deg; joints [71.805, -17.602, 85.459, 0, 22.143, 71.805]
  MoveL 8011 to (-31.5, -51.3, -11.53) mm, rotated rx 180 ry 0 rz 90 deg; joints [71.844, -17.563, 85.372, 0, 22.191, 71.844]
  MoveL 8012 to (-30.4, -50.25, -11.94) mm, rotated rx 180 ry 0 rz 90 deg; joints [71.889, -17.529, 85.306, 0, 22.223, 71.889]
  MoveL 8013 to (-29.56, -48.98, -12.34) mm, rotated rx -180 ry 0 rz 90 deg; joints [71.939, -17.5, 85.262, 0, 22.238, 71.939]
  MoveL 8014 to (-29.05, -47.55, -12.75) mm, rotated rx -180 ry 0 rz 90 deg; joints [71.99, -17.479, 85.245, 0, 22.233, 71.99]
  MoveL 8015 to (-23.66, -26.54, -12.75) mm, rotated rx -180 ry 0 rz 90 deg; joints [72.726, -17.501, 85.335, 0, 22.166, 72.726]
  MoveC 8016 to (-24.4, -24.54, -12.75) mm, rotated rx 180 ry 0 rz 90 deg; joints [72.783, -17.525, 85.429, 0, 22.095, 72.783] to (-26.06, -23.22, -12.75) mm, rotated rx 180 ry 0 rz 90 deg; joints [72.809, -17.561, 85.573, 0, 21.987, 72.809]
  MoveC 8017 to (-26.52, -23.09, -12.75) mm, rotated rx 180 ry 0 rz 90 deg; joints [72.809, -17.57, 85.608, 0, 21.961, 72.809] to (-27.01, -23.11, -12.75) mm, rotated rx 180 ry 0 rz 90 deg; joints [72.803, -17.578, 85.642, 0, 21.936, 72.803]
  MoveC 8018 to (-48.17, -27.33, -12.75) mm, rotated rx 180 ry 0 rz 90 deg; joints [72.449, -17.912, 87.008, 0, 20.904, 72.449] to (-69.32, -31.64, -12.75) mm, rotated rx 180 ry 0 rz 90 deg; joints [72.084, -18.226, 88.347, 0, 19.879, 72.084]
  MoveC 8019 to (-69.71, -31.75, -12.75) mm, rotated rx 180 ry 0 rz 90 deg; joints [72.076, -18.231, 88.371, 0, 19.861, 72.076] to (-70.07, -31.91, -12.75) mm, rotated rx -180 ry 0 rz 90 deg; joints [72.067, -18.236, 88.392, 0, 19.844, 72.067]
  MoveC 8020 to (-71.13, -32.93, -12.75) mm, rotated rx -180 ry 0 rz 90 deg; joints [72.021, -18.248, 88.441, 0, 19.807, 72.021] to (-71.52, -34.36, -12.75) mm, rotated rx -180 ry 0 rz 90 deg; joints [71.97, -18.246, 88.436, 0, 19.81, 71.97]
  MoveL 8021 to (-71.52, -68.39, -12.75) mm, rotated rx 180 ry 0 rz 90 deg; joints [70.849, -18.068, 87.668, 0, 20.401, 70.849]
  MoveC 8022 to (-70.68, -70.4, -12.75) mm, rotated rx 180 ry 0 rz 90 deg; joints [70.793, -18.044, 87.564, 0, 20.48, 70.793] to (-68.66, -71.21, -12.75) mm, rotated rx 180 ry 0 rz 90 deg; joints [70.79, -18.007, 87.409, 0, 20.598, 70.79]
  MoveC 8023 to (-52.91, -70.96, -12.75) mm, rotated rx 180 ry 0 rz 90 deg; joints [70.975, -17.752, 86.348, 0, 21.404, 70.975] to (-37.16, -70.65, -12.75) mm, rotated rx -180 ry 0 rz 90 deg; joints [71.159, -17.486, 85.274, 0, 22.212, 71.159]
  MoveC 8024 to (-35.46, -70.04, -12.75) mm, rotated rx -180 ry 0 rz 90 deg; joints [71.198, -17.46, 85.17, 0, 22.289, 71.198] to (-34.46, -68.54, -12.75) mm, rotated rx 180 ry 0 rz 90 deg; joints [71.257, -17.451, 85.137, 0, 22.315, 71.257]
  MoveL 8025 to (-34.24, -67.76, -12.75) mm, rotated rx 180 ry 0 rz 90 deg; joints [71.284, -17.452, 85.14, 0, 22.312, 71.284]
  MoveL 8026 to (-29.05, -47.55, -12.75) mm, rotated rx -180 ry 0 rz 90 deg; joints [71.99, -17.479, 85.245, 0, 22.233, 71.99]
  MoveL 8027 to (-36.37, -45.67, -12.75) mm, rotated rx 180 ry 0 rz 90 deg; joints [71.974, -17.616, 85.794, 0, 21.822, 71.974]
  MoveL 8028 to (-36.37, -45.67, -9.75) mm, rotated rx 180 ry 0 rz 90 deg; joints [71.974, -17.77, 85.896, 0, 21.874, 71.974]
  Establecer velocidad (1000.0 mm/s)
  MoveL 8029 to (-36.37, -45.67, 10) mm, rotated rx 180 ry 0 rz 90 deg; joints [71.974, -18.787, 86.558, 0, 22.229, 71.974]
  Establecer velocidad (66.7 mm/s)
  MoveL 8030 to (15.02, -45.83, 10) mm, rotated rx -180 ry 0 rz 90 deg; joints [72.496, -17.828, 82.934, 0, 24.894, 72.496]
  MoveL 8031 to (15.02, -45.83, -9.5) mm, rotated rx -180 ry 0 rz 90 deg; joints [72.496, -16.839, 82.279, 0, 24.56, 72.496]
  MoveL 8032 to (13.62, -45.26, -9.91) mm, rotated rx 180 ry 0 rz 90 deg; joints [72.5, -16.849, 82.379, 0, 24.47, 72.5]
  MoveL 8033 to (12.12, -45.03, -10.31) mm, rotated rx -180 ry 0 rz 90 deg; joints [72.492, -16.859, 82.478, 0, 24.381, 72.492]
  MoveL 8034 to (10.6, -45.15, -10.72) mm, rotated rx 180 ry 0 rz 90 deg; joints [72.473, -16.867, 82.571, 0, 24.297, 72.473]
  MoveL 8035 to (9.15, -45.6, -11.13) mm, rotated rx 180 ry 0 rz 90 deg; joints [72.444, -16.872, 82.65, 0, 24.221, 72.444]
  MoveL 8036 to (7.83, -46.36, -11.53) mm, rotated rx 180 ry 0 rz 90 deg; joints [72.407, -16.872, 82.714, 0, 24.158, 72.407]
  MoveL 8037 to (6.72, -47.39, -11.94) mm, rotated rx 180 ry 0 rz 90 deg; joints [72.363, -16.866, 82.756, 0, 24.11, 72.363]
  MoveL 8038 to (5.86, -48.64, -12.34) mm, rotated rx -180 ry 0 rz 90 deg; joints [72.315, -16.854, 82.775, 0, 24.079, 72.315]
  MoveL 8039 to (5.33, -50.06, -12.75) mm, rotated rx 180 ry 0 rz 90 deg; joints [72.264, -16.835, 82.767, 0, 24.068, 72.264]
  MoveL 8040 to (0.89, -66.31, -12.75) mm, rotated rx -180 ry 0 rz 90 deg; joints [71.705, -16.819, 82.707, 0, 24.112, 71.705]
  MoveC 8041 to (0.83, -67.14, -12.75) mm, rotated rx -180 ry 0 rz 90 deg; joints [71.678, -16.815, 82.691, 0, 24.124, 71.678] to (1.09, -67.93, -12.75) mm, rotated rx 180 ry 0 rz 90 deg; joints [71.656, -16.805, 82.654, 0, 24.151, 71.656]
  MoveL 8042 to (1.3, -68.3, -12.75) mm, rotated rx -180 ry 0 rz 90 deg; joints [71.646, -16.799, 82.631, 0, 24.168, 71.646]
  MoveC 8043 to (2.41, -69.41, -12.75) mm, rotated rx 180 ry 0 rz 90 deg; joints [71.623, -16.77, 82.524, 0, 24.246, 71.623] to (3.95, -69.78, -12.75) mm, rotated rx 180 ry 0 rz 90 deg; joints [71.627, -16.738, 82.406, 0, 24.332, 71.627]
  MoveC 8044 to (14.67, -69.37, -12.75) mm, rotated rx 180 ry 0 rz 90 deg; joints [71.752, -16.532, 81.646, 0, 24.886, 71.752] to (25.39, -68.84, -12.75) mm, rotated rx -180 ry 0 rz 90 deg; joints [71.878, -16.321, 80.881, 0, 25.439, 71.878]
  MoveL 8045 to (25.39, -43.9, -12.75) mm, rotated rx 180 ry 0 rz 90 deg; joints [72.659, -16.481, 81.462, 0, 25.019, 72.659]
  MoveL 8046 to (22.43, -40.27, -12.75) mm, rotated rx 180 ry 0 rz 90 deg; joints [72.744, -16.562, 81.758, 0, 24.804, 72.744]
  MoveL 8047 to (22.27, -40.1, -12.75) mm, rotated rx 180 ry 0 rz 90 deg; joints [72.748, -16.567, 81.774, 0, 24.793, 72.748]
  MoveL 8048 to (21.4, -39.33, -12.75) mm, rotated rx 180 ry 0 rz 90 deg; joints [72.764, -16.589, 81.854, 0, 24.734, 72.764]
  MoveL 8049 to (14.61, -33.64, -12.75) mm, rotated rx 180 ry 0 rz 90 deg; joints [72.878, -16.756, 82.471, 0, 24.285, 72.878]
  MoveL 8050 to (14.21, -33.31, -12.75) mm, rotated rx -180 ry 0 rz 90 deg; joints [72.884, -16.765, 82.507, 0, 24.259, 72.884]
  MoveC 8051 to (11.99, -32.92, -12.75) mm, rotated rx -180 ry 0 rz 90 deg; joints [72.875, -16.811, 82.675, 0, 24.135, 72.875] to (9.95, -33.89, -12.75) mm, rotated rx 180 ry 0 rz 90 deg; joints [72.824, -16.844, 82.8, 0, 24.044, 72.824]
  MoveL 8052 to (9.81, -34.06, -12.75) mm, rotated rx -180 ry 0 rz 90 deg; joints [72.817, -16.846, 82.806, 0, 24.04, 72.817]
  MoveL 8053 to (9.48, -34.88, -12.75) mm, rotated rx -180 ry 0 rz 90 deg; joints [72.788, -16.847, 82.812, 0, 24.035, 72.788]
  MoveL 8054 to (5.33, -50.06, -12.75) mm, rotated rx 180 ry 0 rz 90 deg; joints [72.264, -16.835, 82.767, 0, 24.068, 72.264]
  MoveL 8055 to (12.61, -52.05, -12.75) mm, rotated rx -180 ry 0 rz 90 deg; joints [72.275, -16.682, 82.199, 0, 24.483, 72.275]
  MoveL 8056 to (12.61, -52.05, -9.75) mm, rotated rx 180 ry 0 rz 90 deg; joints [72.275, -16.835, 82.302, 0, 24.533, 72.275]
  Establecer velocidad (1000.0 mm/s)
  MoveL 8057 to (12.61, -52.05, 10) mm, rotated rx -180 ry 0 rz 90 deg; joints [72.275, -17.837, 82.966, 0, 24.871, 72.275]
  Establecer velocidad (66.7 mm/s)
  MoveL 8058 to (14.43, 20.21, 10) mm, rotated rx 180 ry 0 rz 90 deg; joints [74.6, -18.219, 84.377, 0, 23.842, 74.6]
  MoveL 8059 to (14.43, 20.21, -9.5) mm, rotated rx -180 ry 0 rz 90 deg; joints [74.6, -17.225, 83.723, 0, 23.502, 74.6]
  MoveL 8060 to (14.18, 18.71, -9.91) mm, rotated rx 180 ry 0 rz 90 deg; joints [74.55, -17.201, 83.697, 0, 23.504, 74.55]
  MoveL 8061 to (14.38, 17.21, -10.31) mm, rotated rx 180 ry 0 rz 90 deg; joints [74.503, -17.169, 83.64, 0, 23.529, 74.503]
  MoveL 8062 to (14.96, 15.81, -10.72) mm, rotated rx 180 ry 0 rz 90 deg; joints [74.463, -17.13, 83.556, 0, 23.574, 74.463]
  MoveL 8063 to (15.91, 14.62, -11.13) mm, rotated rx 180 ry 0 rz 90 deg; joints [74.433, -17.085, 83.451, 0, 23.634, 74.433]
  MoveL 8064 to (17.13, 13.72, -11.53) mm, rotated rx 180 ry 0 rz 90 deg; joints [74.415, -17.036, 83.331, 0, 23.706, 74.415]
  MoveL 8065 to (18.55, 13.19, -11.94) mm, rotated rx -180 ry 0 rz 90 deg; joints [74.411, -16.986, 83.204, 0, 23.782, 74.411]
  MoveL 8066 to (20.07, 13.05, -12.34) mm, rotated rx 180 ry 0 rz 90 deg; joints [74.42, -16.935, 83.078, 0, 23.857, 74.42]
  MoveL 8067 to (21.55, 13.36, -12.75) mm, rotated rx -180 ry 0 rz 90 deg; joints [74.443, -16.888, 82.963, 0, 23.924, 74.443]
  MoveL 8068 to (25.39, 14.62, -12.75) mm, rotated rx -180 ry 0 rz 90 deg; joints [74.518, -16.82, 82.712, 0, 24.109, 74.518]
  MoveL 8069 to (25.39, 24.26, -12.75) mm, rotated rx 180 ry 0 rz 90 deg; joints [74.827, -16.872, 82.903, 0, 23.969, 74.827]
  MoveL 8070 to (16.58, 24.34, -12.75) mm, rotated rx 180 ry 0 rz 90 deg; joints [74.753, -17.04, 83.539, 0, 23.501, 74.753]
  MoveL 8071 to (15.64, 24.31, -12.75) mm, rotated rx -180 ry 0 rz 90 deg; joints [74.743, -17.057, 83.606, 0, 23.451, 74.743]
  MoveC 8072 to (13.62, 23.11, -12.75) mm, rotated rx -180 ry 0 rz 90 deg; joints [74.687, -17.089, 83.727, 0, 23.362, 74.687] to (13.03, 20.85, -12.75) mm, rotated rx 180 ry 0 rz 90 deg; joints [74.608, -17.089, 83.725, 0, 23.364, 74.608]
  MoveL 8073 to (16.25, 12.2, -12.75) mm, rotated rx -180 ry 0 rz 90 deg; joints [74.358, -16.983, 83.322, 0, 23.661, 74.358]
  MoveC 8074 to (16.62, 11.52, -12.75) mm, rotated rx 180 ry 0 rz 90 deg; joints [74.34, -16.972, 83.281, 0, 23.691, 74.34] to (17.18, 10.97, -12.75) mm, rotated rx -180 ry 0 rz 90 deg; joints [74.327, -16.958, 83.23, 0, 23.728, 74.327]
  MoveL 8075 to (18.48, 10.01, -12.75) mm, rotated rx -180 ry 0 rz 90 deg; joints [74.308, -16.929, 83.117, 0, 23.811, 74.308]
  MoveL 8076 to (24.17, 5.86, -12.75) mm, rotated rx 180 ry 0 rz 90 deg; joints [74.226, -16.797, 82.623, 0, 24.174, 74.226]
  MoveL 8077 to (25.39, 4.99, -12.75) mm, rotated rx 180 ry 0 rz 90 deg; joints [74.209, -16.768, 82.517, 0, 24.251, 74.209]
  MoveL 8078 to (25.39, 14.62, -12.75) mm, rotated rx -180 ry 0 rz 90 deg; joints [74.518, -16.82, 82.712, 0, 24.109, 74.518]
  MoveL 8079 to (17.84, 14.62, -12.75) mm, rotated rx 180 ry 0 rz 90 deg; joints [74.45, -16.965, 83.256, 0, 23.709, 74.45]
  MoveL 8080 to (17.84, 14.62, -9.75) mm, rotated rx 180 ry 0 rz 90 deg; joints [74.45, -17.118, 83.359, 0, 23.76, 74.45]
  Establecer velocidad (1000.0 mm/s)
  MoveL 8081 to (17.84, 14.62, 10) mm, rotated rx -180 ry 0 rz 90 deg; joints [74.45, -18.124, 84.022, 0, 24.103, 74.45]
  Establecer velocidad (66.7 mm/s)
  MoveL 8082 to (-7.72, 66.16, 10) mm, rotated rx -180 ry 0 rz 90 deg; joints [75.913, -18.849, 86.804, 0, 22.044, 75.913]
  MoveL 8083 to (-7.72, 66.16, -9.5) mm, rotated rx 180 ry 0 rz 90 deg; joints [75.913, -17.844, 86.151, 0, 21.693, 75.913]
  MoveL 8084 to (-8.14, 64.7, -9.91) mm, rotated rx -180 ry 0 rz 90 deg; joints [75.861, -17.824, 86.141, 0, 21.683, 75.861]
  MoveL 8085 to (-8.15, 63.19, -10.31) mm, rotated rx -180 ry 0 rz 90 deg; joints [75.81, -17.797, 86.101, 0, 21.696, 75.81]
  MoveL 8086 to (-7.76, 61.71, -10.72) mm, rotated rx -180 ry 0 rz 90 deg; joints [75.765, -17.763, 86.034, 0, 21.728, 75.765]
  MoveL 8087 to (-7.02, 60.39, -11.13) mm, rotated rx -180 ry 0 rz 90 deg; joints [75.727, -17.723, 85.945, 0, 21.778, 75.727]
  MoveL 8088 to (-5.97, 59.29, -11.53) mm, rotated rx 180 ry 0 rz 90 deg; joints [75.7, -17.679, 85.837, 0, 21.842, 75.7]
  MoveL 8089 to (-4.67, 58.51, -11.94) mm, rotated rx 180 ry 0 rz 90 deg; joints [75.685, -17.632, 85.718, 0, 21.914, 75.685]
  MoveL 8090 to (-3.21, 58.07, -12.34) mm, rotated rx -180 ry 0 rz 90 deg; joints [75.683, -17.583, 85.593, 0, 21.99, 75.683]
  MoveL 8091 to (-1.7, 58.06, -12.75) mm, rotated rx 180 ry 0 rz 90 deg; joints [75.695, -17.536, 85.472, 0, 22.063, 75.695]
  MoveL 8092 to (4.43, 58.66, -12.75) mm, rotated rx 180 ry 0 rz 90 deg; joints [75.766, -17.429, 85.05, 0, 22.379, 75.766]
  MoveC 8093 to (14.92, 59.82, -12.75) mm, rotated rx -180 ry 0 rz 90 deg; joints [75.891, -17.244, 84.324, 0, 22.92, 75.891] to (25.39, 61.15, -12.75) mm, rotated rx 180 ry 0 rz 90 deg; joints [76.02, -17.055, 83.596, 0, 23.459, 76.02]
  MoveL 8094 to (25.39, 68.65, -12.75) mm, rotated rx -180 ry 0 rz 90 deg; joints [76.264, -17.09, 83.729, 0, 23.361, 76.264]
  MoveC 8095 to (6.26, 69.5, -12.75) mm, rotated rx 180 ry 0 rz 90 deg; joints [76.138, -17.445, 85.112, 0, 22.333, 76.138] to (-12.87, 70.13, -12.75) mm, rotated rx 180 ry 0 rz 90 deg; joints [76.001, -17.782, 86.471, 0, 21.311, 76.001]
  MoveC 8096 to (-14.91, 67.59, -12.75) mm, rotated rx 180 ry 0 rz 90 deg; joints [75.9, -17.806, 86.569, 0, 21.237, 75.9] to (-14.67, 64.34, -12.75) mm, rotated rx 180 ry 0 rz 90 deg; joints [75.794, -17.788, 86.495, 0, 21.293, 75.794]
  MoveL 8097 to (-6.87, 59.23, -12.75) mm, rotated rx -180 ry 0 rz 90 deg; joints [75.69, -17.631, 85.858, 0, 21.774, 75.69]
  MoveL 8098 to (-5.19, 58.07, -12.75) mm, rotated rx 180 ry 0 rz 90 deg; joints [75.666, -17.597, 85.719, 0, 21.878, 75.666]
  MoveC 8099 to (-4.93, 57.92, -12.75) mm, rotated rx -180 ry 0 rz 90 deg; joints [75.663, -17.592, 85.698, 0, 21.894, 75.663] to (-4.67, 57.79, -12.75) mm, rotated rx 180 ry 0 rz 90 deg; joints [75.661, -17.587, 85.677, 0, 21.91, 75.661]
  MoveC 8100 to (-0.12, 58.21, -12.75) mm, rotated rx -180 ry 0 rz 90 deg; joints [75.713, -17.508, 85.364, 0, 22.145, 75.713] to (4.43, 58.66, -12.75) mm, rotated rx 180 ry 0 rz 90 deg; joints [75.766, -17.429, 85.05, 0, 22.379, 75.766]
  MoveL 8101 to (3.66, 66.17, -12.75) mm, rotated rx -180 ry 0 rz 90 deg; joints [76.007, -17.477, 85.238, 0, 22.238, 76.007]
  MoveL 8102 to (3.66, 66.17, -9.75) mm, rotated rx -180 ry 0 rz 90 deg; joints [76.007, -17.631, 85.341, 0, 22.29, 76.007]
  Establecer velocidad (1000.0 mm/s)
  MoveL 8103 to (3.66, 66.17, 10) mm, rotated rx 180 ry 0 rz 90 deg; joints [76.007, -18.645, 86.003, 0, 22.642, 76.007]
  Establecer velocidad (66.7 mm/s)
  MoveL 8104 to (-63.28, 35.68, 10) mm, rotated rx 180 ry 0 rz 90 deg; joints [74.399, -19.632, 90.069, 0, 19.563, 74.399]
  MoveL 8105 to (-63.28, 35.68, -9.5) mm, rotated rx 180 ry 0 rz 90 deg; joints [74.399, -18.613, 89.416, 0, 19.197, 74.399]
  MoveL 8106 to (-64.79, 35.87, -9.91) mm, rotated rx 180 ry 0 rz 90 deg; joints [74.391, -18.615, 89.507, 0, 19.108, 74.391]
  MoveL 8107 to (-66.3, 35.69, -10.31) mm, rotated rx 180 ry 0 rz 90 deg; joints [74.371, -18.615, 89.591, 0, 19.024, 74.371]
  MoveL 8108 to (-67.73, 35.18, -10.72) mm, rotated rx 180 ry 0 rz 90 deg; joints [74.34, -18.613, 89.664, 0, 18.95, 74.34]
  MoveL 8109 to (-69.01, 34.36, -11.13) mm, rotated rx 180 ry 0 rz 90 deg; joints [74.3, -18.608, 89.72, 0, 18.887, 74.3]
  MoveL 8110 to (-70.08, 33.28, -11.53) mm, rotated rx 180 ry 0 rz 90 deg; joints [74.253, -18.598, 89.758, 0, 18.84, 74.253]
  MoveL 8111 to (-70.88, 31.99, -11.94) mm, rotated rx -180 ry 0 rz 90 deg; joints [74.202, -18.583, 89.773, 0, 18.809, 74.202]
  MoveL 8112 to (-71.38, 30.56, -12.34) mm, rotated rx 180 ry 0 rz 90 deg; joints [74.148, -18.563, 89.766, 0, 18.797, 74.148]
  MoveL 8113 to (-71.52, 29.04, -12.75) mm, rotated rx 180 ry 0 rz 90 deg; joints [74.096, -18.537, 89.732, 0, 18.805, 74.096]
  MoveL 8114 to (-71.52, 3.84, -12.75) mm, rotated rx -180 ry 0 rz 90 deg; joints [73.245, -18.428, 89.238, 0, 19.19, 73.245]
  MoveC 8115 to (-71.01, 2.2, -12.75) mm, rotated rx -180 ry 0 rz 90 deg; joints [73.195, -18.413, 89.171, 0, 19.242, 73.195] to (-69.65, 1.15, -12.75) mm, rotated rx -180 ry 0 rz 90 deg; joints [73.174, -18.388, 89.058, 0, 19.329, 73.174]
  MoveC 8116 to (-68.91, 0.96, -12.75) mm, rotated rx 180 ry 0 rz 90 deg; joints [73.175, -18.375, 89.004, 0, 19.371, 73.175] to (-68.14, 1.01, -12.75) mm, rotated rx -180 ry 0 rz 90 deg; joints [73.184, -18.364, 88.954, 0, 19.41, 73.184]
  MoveC 8117 to (-46.45, 6.18, -12.75) mm, rotated rx 180 ry 0 rz 90 deg; joints [73.573, -18.05, 87.59, 0, 20.46, 73.573] to (-24.79, 11.46, -12.75) mm, rotated rx 180 ry 0 rz 90 deg; joints [73.955, -17.717, 86.204, 0, 21.513, 73.955]
  MoveC 8118 to (-23.9, 11.87, -12.75) mm, rotated rx 180 ry 0 rz 90 deg; joints [73.977, -17.704, 86.15, 0, 21.553, 73.977] to (-23.22, 12.57, -12.75) mm, rotated rx 180 ry 0 rz 90 deg; joints [74.007, -17.695, 86.117, 0, 21.578, 74.007]
  MoveC 8119 to (-22.62, 13.98, -12.75) mm, rotated rx 180 ry 0 rz 90 deg; joints [74.058, -17.692, 86.104, 0, 21.588, 74.058] to (-22.77, 15.5, -12.75) mm, rotated rx -180 ry 0 rz 90 deg; joints [74.107, -17.702, 86.144, 0, 21.558, 74.107]
  MoveL 8120 to (-27.93, 30.1, -12.75) mm, rotated rx -180 ry 0 rz 90 deg; joints [74.541, -17.858, 86.786, 0, 21.072, 74.541]
  MoveC 8121 to (-28.44, 31.03, -12.75) mm, rotated rx 180 ry 0 rz 90 deg; joints [74.567, -17.871, 86.839, 0, 21.032, 74.567] to (-29.21, 31.74, -12.75) mm, rotated rx 180 ry 0 rz 90 deg; joints [74.584, -17.887, 86.907, 0, 20.981, 74.584]
  MoveC 8122 to (-48.22, 44.22, -12.75) mm, rotated rx -180 ry 0 rz 90 deg; joints [74.827, -18.248, 88.445, 0, 19.804, 74.827] to (-67.28, 56.62, -12.75) mm, rotated rx -180 ry 0 rz 90 deg; joints [75.074, -18.586, 89.958, 0, 18.629, 75.074]
  MoveC 8123 to (-67.74, 56.81, -12.75) mm, rotated rx 180 ry 0 rz 90 deg; joints [75.076, -18.594, 89.992, 0, 18.602, 75.076] to (-68.23, 56.86, -12.75) mm, rotated rx 180 ry 0 rz 90 deg; joints [75.073, -18.601, 90.025, 0, 18.576, 75.073]
  MoveC 8124 to (-69.84, 56.47, -12.75) mm, rotated rx 180 ry 0 rz 90 deg; joints [75.045, -18.623, 90.127, 0, 18.496, 75.045] to (-71.13, 55.41, -12.75) mm, rotated rx 180 ry 0 rz 90 deg; joints [74.997, -18.638, 90.193, 0, 18.444, 74.997]
  MoveC 8125 to (-71.42, 54.86, -12.75) mm, rotated rx 180 ry 0 rz 90 deg; joints [74.976, -18.64, 90.203, 0, 18.437, 74.976] to (-71.52, 54.25, -12.75) mm, rotated rx 180 ry 0 rz 90 deg; joints [74.954, -18.639, 90.199, 0, 18.44, 74.954]
  MoveL 8126 to (-71.52, 29.04, -12.75) mm, rotated rx 180 ry 0 rz 90 deg; joints [74.096, -18.537, 89.732, 0, 18.805, 74.096]
  MoveL 8127 to (-63.97, 29.04, -12.75) mm, rotated rx -180 ry 0 rz 90 deg; joints [74.168, -18.425, 89.226, 0, 19.199, 74.168]
  MoveL 8128 to (-63.97, 29.04, -9.75) mm, rotated rx 180 ry 0 rz 90 deg; joints [74.168, -18.582, 89.328, 0, 19.254, 74.168]
  Establecer velocidad (1000.0 mm/s)
  MoveL 8129 to (-63.97, 29.04, 10) mm, rotated rx 180 ry 0 rz 90 deg; joints [74.168, -19.614, 89.99, 0, 19.624, 74.168]
  Establecer velocidad (66.7 mm/s)
  MoveL 8130 to (-63.12, 35.68, 10) mm, rotated rx -180 ry 0 rz 90 deg; joints [74.401, -19.63, 90.058, 0, 19.571, 74.401]
  MoveL 8131 to (-63.12, 35.68, -9.75) mm, rotated rx 180 ry 0 rz 90 deg; joints [74.401, -18.597, 89.396, 0, 19.201, 74.401]
  MoveL 8132 to (-64.63, 35.87, -10.16) mm, rotated rx -180 ry 0 rz 90 deg; joints [74.393, -18.599, 89.487, 0, 19.112, 74.393]
  MoveL 8133 to (-66.13, 35.69, -10.56) mm, rotated rx -180 ry 0 rz 90 deg; joints [74.372, -18.6, 89.572, 0, 19.028, 74.372]
  MoveL 8134 to (-67.56, 35.18, -10.97) mm, rotated rx 180 ry 0 rz 90 deg; joints [74.342, -18.598, 89.644, 0, 18.954, 74.342]
  MoveL 8135 to (-68.85, 34.36, -11.37) mm, rotated rx 180 ry 0 rz 90 deg; joints [74.302, -18.592, 89.701, 0, 18.891, 74.302]
  MoveL 8136 to (-69.92, 33.28, -11.78) mm, rotated rx 180 ry 0 rz 90 deg; joints [74.255, -18.582, 89.738, 0, 18.844, 74.255]
  MoveL 8137 to (-70.72, 31.99, -12.19) mm, rotated rx 180 ry 0 rz 90 deg; joints [74.203, -18.567, 89.754, 0, 18.813, 74.203]
  MoveL 8138 to (-71.22, 30.56, -12.59) mm, rotated rx 180 ry 0 rz 90 deg; joints [74.15, -18.547, 89.746, 0, 18.801, 74.15]
  MoveL 8139 to (-71.36, 29.04, -13) mm, rotated rx -180 ry 0 rz 90 deg; joints [74.097, -18.522, 89.713, 0, 18.809, 74.097]
  MoveL 8140 to (-71.36, 3.98, -13) mm, rotated rx -180 ry 0 rz 90 deg; joints [73.251, -18.413, 89.221, 0, 19.192, 73.251]
  MoveC 8141 to (-70.28, 1.75, -13) mm, rotated rx -180 ry 0 rz 90 deg; joints [73.187, -18.387, 89.104, 0, 19.283, 73.187] to (-67.87, 1.22, -13) mm, rotated rx -180 ry 0 rz 90 deg; joints [73.194, -18.348, 88.932, 0, 19.416, 73.194]
  MoveC 8142 to (-46.48, 6.34, -13) mm, rotated rx -180 ry 0 rz 90 deg; joints [73.577, -18.038, 87.587, 0, 20.452, 73.577] to (-25.11, 11.55, -13) mm, rotated rx -180 ry 0 rz 90 deg; joints [73.955, -17.71, 86.22, 0, 21.49, 73.955]
  MoveC 8143 to (-24, 12.06, -13) mm, rotated rx 180 ry 0 rz 90 deg; joints [73.983, -17.693, 86.153, 0, 21.541, 73.983] to (-23.22, 13.01, -13) mm, rotated rx 180 ry 0 rz 90 deg; joints [74.021, -17.685, 86.118, 0, 21.567, 74.021]
  MoveC 8144 to (-22.8, 14.3, -13) mm, rotated rx 180 ry 0 rz 90 deg; joints [74.067, -17.684, 86.114, 0, 21.57, 74.067] to (-22.98, 15.64, -13) mm, rotated rx 180 ry 0 rz 90 deg; joints [74.11, -17.694, 86.153, 0, 21.54, 74.11]
  MoveL 8145 to (-28.07, 30.03, -13) mm, rotated rx 180 ry 0 rz 90 deg; joints [74.538, -17.847, 86.786, 0, 21.061, 74.538]
  MoveC 8146 to (-28.55, 30.92, -13) mm, rotated rx -180 ry 0 rz 90 deg; joints [74.563, -17.86, 86.837, 0, 21.023, 74.563] to (-29.3, 31.61, -13) mm, rotated rx -180 ry 0 rz 90 deg; joints [74.579, -17.875, 86.901, 0, 20.974, 74.579]
  MoveC 8147 to (-48.21, 44.03, -13) mm, rotated rx -180 ry 0 rz 90 deg; joints [74.821, -18.234, 88.432, 0, 19.803, 74.821] to (-67.16, 56.39, -13) mm, rotated rx 180 ry 0 rz 90 deg; joints [75.067, -18.571, 89.937, 0, 18.634, 75.067]
  MoveC 8148 to (-67.45, 56.53, -13) mm, rotated rx -180 ry 0 rz 90 deg; joints [75.069, -18.575, 89.958, 0, 18.617, 75.069] to (-67.76, 56.58, -13) mm, rotated rx 180 ry 0 rz 90 deg; joints [75.068, -18.58, 89.98, 0, 18.6, 75.068]
  MoveC 8149 to (-69.63, 56.26, -13) mm, rotated rx 180 ry 0 rz 90 deg; joints [75.04, -18.606, 90.1, 0, 18.506, 75.04] to (-71.07, 55.02, -13) mm, rotated rx -180 ry 0 rz 90 deg; joints [74.984, -18.622, 90.174, 0, 18.448, 74.984]
  MoveC 8150 to (-71.28, 54.56, -13) mm, rotated rx -180 ry 0 rz 90 deg; joints [74.967, -18.623, 90.18, 0, 18.443, 74.967] to (-71.36, 54.07, -13) mm, rotated rx -180 ry 0 rz 90 deg; joints [74.949, -18.623, 90.176, 0, 18.446, 74.949]
  MoveL 8151 to (-71.36, 29.04, -13) mm, rotated rx -180 ry 0 rz 90 deg; joints [74.097, -18.522, 89.713, 0, 18.809, 74.097]
  MoveL 8152 to (-63.81, 29.04, -13) mm, rotated rx -180 ry 0 rz 90 deg; joints [74.17, -18.41, 89.206, 0, 19.204, 74.17]
  MoveL 8153 to (-63.81, 29.04, -10) mm, rotated rx 180 ry 0 rz 90 deg; joints [74.17, -18.566, 89.309, 0, 19.258, 74.17]
  Establecer velocidad (1000.0 mm/s)
  MoveL 8154 to (-63.81, 29.04, 10) mm, rotated rx 180 ry 0 rz 90 deg; joints [74.17, -19.612, 89.979, 0, 19.633, 74.17]
  Establecer velocidad (66.7 mm/s)
  MoveL 8155 to (-6.49, 59.94, 10) mm, rotated rx 180 ry 0 rz 90 deg; joints [75.717, -18.799, 86.608, 0, 22.191, 75.717]
  MoveL 8156 to (-6.49, 59.94, -9.75) mm, rotated rx -180 ry 0 rz 90 deg; joints [75.717, -17.783, 85.946, 0, 21.836, 75.717]
  MoveL 8157 to (-5.33, 58.96, -10.16) mm, rotated rx 180 ry 0 rz 90 deg; joints [75.694, -17.737, 85.833, 0, 21.904, 75.694]
  MoveL 8158 to (-3.95, 58.34, -10.56) mm, rotated rx -180 ry 0 rz 90 deg; joints [75.686, -17.689, 85.711, 0, 21.978, 75.686]
  MoveL 8159 to (-2.44, 58.11, -10.97) mm, rotated rx -180 ry 0 rz 90 deg; joints [75.691, -17.641, 85.587, 0, 22.054, 75.691]
  MoveL 8160 to (-0.93, 58.28, -11.37) mm, rotated rx 180 ry 0 rz 90 deg; joints [75.709, -17.594, 85.47, 0, 22.124, 75.709]
  MoveL 8161 to (0.48, 58.84, -11.78) mm, rotated rx 180 ry 0 rz 90 deg; joints [75.739, -17.55, 85.366, 0, 22.185, 75.739]
  MoveL 8162 to (1.7, 59.75, -12.19) mm, rotated rx 180 ry 0 rz 90 deg; joints [75.779, -17.512, 85.282, 0, 22.23, 75.779]
  MoveL 8163 to (2.64, 60.94, -12.59) mm, rotated rx 180 ry 0 rz 90 deg; joints [75.826, -17.48, 85.223, 0, 22.257, 75.826]
  MoveL 8164 to (3.21, 62.35, -13) mm, rotated rx -180 ry 0 rz 90 deg; joints [75.877, -17.455, 85.194, 0, 22.261, 75.877]
  MoveL 8165 to (5.15, 69.34, -13) mm, rotated rx -180 ry 0 rz 90 deg; joints [76.124, -17.452, 85.18, 0, 22.271, 76.124]
  MoveC 8166 to (-3.55, 69.66, -13) mm, rotated rx -180 ry 0 rz 90 deg; joints [76.063, -17.606, 85.8, 0, 21.806, 76.063] to (-12.25, 69.93, -13) mm, rotated rx 180 ry 0 rz 90 deg; joints [76, -17.758, 86.415, 0, 21.342, 76]
  MoveC 8167 to (-14.26, 67.42, -13) mm, rotated rx 180 ry 0 rz 90 deg; joints [75.9, -17.781, 86.512, 0, 21.269, 75.9] to (-14.04, 64.21, -13) mm, rotated rx -180 ry 0 rz 90 deg; joints [75.795, -17.764, 86.44, 0, 21.324, 75.795]
  MoveL 8168 to (-6.46, 59.23, -13) mm, rotated rx -180 ry 0 rz 90 deg; joints [75.694, -17.611, 85.82, 0, 21.791, 75.694]
  MoveL 8169 to (-4.79, 58.06, -13) mm, rotated rx -180 ry 0 rz 90 deg; joints [75.669, -17.577, 85.682, 0, 21.895, 75.669]
  MoveC 8170 to (-4.55, 57.95, -13) mm, rotated rx -180 ry 0 rz 90 deg; joints [75.668, -17.572, 85.663, 0, 21.909, 75.668] to (-4.3, 57.92, -13) mm, rotated rx 180 ry 0 rz 90 deg; joints [75.669, -17.568, 85.645, 0, 21.923, 75.669]
  MoveC 8171 to (9.13, 59.31, -13) mm, rotated rx 180 ry 0 rz 90 deg; joints [75.827, -17.335, 84.719, 0, 22.616, 75.827] to (22.53, 60.93, -13) mm, rotated rx -180 ry 0 rz 90 deg; joints [75.989, -17.095, 83.789, 0, 23.306, 75.989]
  MoveL 8172 to (22.53, 68.56, -13) mm, rotated rx -180 ry 0 rz 90 deg; joints [76.238, -17.13, 83.925, 0, 23.205, 76.238]
  MoveC 8173 to (13.84, 68.98, -13) mm, rotated rx 180 ry 0 rz 90 deg; joints [76.182, -17.293, 84.555, 0, 22.738, 76.182] to (5.15, 69.34, -13) mm, rotated rx -180 ry 0 rz 90 deg; joints [76.124, -17.452, 85.18, 0, 22.271, 76.124]
  MoveL 8174 to (4.85, 61.8, -13) mm, rotated rx -180 ry 0 rz 90 deg; joints [75.873, -17.423, 85.068, 0, 22.355, 75.873]
  MoveL 8175 to (4.85, 61.8, -10) mm, rotated rx 180 ry 0 rz 90 deg; joints [75.873, -17.577, 85.17, 0, 22.407, 75.873]
  Establecer velocidad (1000.0 mm/s)
  MoveL 8176 to (4.85, 61.8, 10) mm, rotated rx -180 ry 0 rz 90 deg; joints [75.873, -18.603, 85.841, 0, 22.763, 75.873]
  Establecer velocidad (66.7 mm/s)
  MoveL 8177 to (19.47, 9.58, 10) mm, rotated rx -180 ry 0 rz 90 deg; joints [74.303, -18.065, 83.803, 0, 24.262, 74.303]
  MoveL 8178 to (19.47, 9.58, -9.75) mm, rotated rx -180 ry 0 rz 90 deg; joints [74.303, -17.06, 83.14, 0, 23.92, 74.303]
  MoveL 8179 to (22.53, 7.36, -10.76) mm, rotated rx 180 ry 0 rz 90 deg; joints [74.259, -16.938, 82.84, 0, 24.098, 74.259]
  MoveL 8180 to (22.53, 15.71, -13) mm, rotated rx 180 ry 0 rz 90 deg; joints [74.527, -16.869, 82.931, 0, 23.937, 74.527]
  MoveL 8181 to (22.53, 24.06, -13) mm, rotated rx 180 ry 0 rz 90 deg; joints [74.796, -16.913, 83.097, 0, 23.816, 74.796]
  MoveL 8182 to (16.58, 24.12, -13) mm, rotated rx 180 ry 0 rz 90 deg; joints [74.746, -17.026, 83.526, 0, 23.5, 74.746]
  MoveL 8183 to (15.64, 24.05, -13) mm, rotated rx -180 ry 0 rz 90 deg; joints [74.735, -17.043, 83.592, 0, 23.451, 74.735]
  MoveC 8184 to (13.9, 22.87, -13) mm, rotated rx 180 ry 0 rz 90 deg; joints [74.681, -17.07, 83.694, 0, 23.376, 74.681] to (13.3, 20.85, -13) mm, rotated rx -180 ry 0 rz 90 deg; joints [74.611, -17.071, 83.697, 0, 23.374, 74.611]
  MoveL 8185 to (13.45, 20.37, -13) mm, rotated rx 180 ry 0 rz 90 deg; joints [74.597, -17.065, 83.677, 0, 23.389, 74.597]
  MoveL 8186 to (16.43, 12.39, -13) mm, rotated rx 180 ry 0 rz 90 deg; joints [74.366, -16.967, 83.304, 0, 23.664, 74.366]
  MoveC 8187 to (16.83, 11.66, -13) mm, rotated rx -180 ry 0 rz 90 deg; joints [74.346, -16.956, 83.261, 0, 23.695, 74.346] to (17.42, 11.08, -13) mm, rotated rx 180 ry 0 rz 90 deg; joints [74.333, -16.942, 83.207, 0, 23.735, 74.333]
  MoveL 8188 to (18.48, 10.3, -13) mm, rotated rx 180 ry 0 rz 90 deg; joints [74.317, -16.917, 83.115, 0, 23.803, 74.317]
  MoveL 8189 to (22.53, 7.36, -13) mm, rotated rx 180 ry 0 rz 90 deg; joints [74.259, -16.824, 82.763, 0, 24.061, 74.259]
  MoveL 8190 to (22.53, 15.71, -13) mm, rotated rx 180 ry 0 rz 90 deg; joints [74.527, -16.869, 82.931, 0, 23.937, 74.527]
  MoveL 8191 to (21.87, 23.23, -13) mm, rotated rx 180 ry 0 rz 90 deg; joints [74.763, -16.921, 83.128, 0, 23.793, 74.763]
  MoveL 8192 to (21.87, 23.23, -10) mm, rotated rx 180 ry 0 rz 90 deg; joints [74.763, -17.074, 83.231, 0, 23.843, 74.763]
  Establecer velocidad (1000.0 mm/s)
  MoveL 8193 to (21.87, 23.23, 10) mm, rotated rx 180 ry 0 rz 90 deg; joints [74.763, -18.092, 83.902, 0, 24.19, 74.763]
  Establecer velocidad (66.7 mm/s)
  MoveL 8194 to (15.18, -46.11, 10) mm, rotated rx 180 ry 0 rz 90 deg; joints [72.488, -17.823, 82.916, 0, 24.907, 72.488]
  MoveL 8195 to (15.18, -46.11, -9.75) mm, rotated rx 180 ry 0 rz 90 deg; joints [72.488, -16.821, 82.252, 0, 24.569, 72.488]
  MoveL 8196 to (13.78, -45.54, -10.16) mm, rotated rx 180 ry 0 rz 90 deg; joints [72.493, -16.832, 82.353, 0, 24.479, 72.493]
  MoveL 8197 to (12.28, -45.32, -10.56) mm, rotated rx 180 ry 0 rz 90 deg; joints [72.485, -16.842, 82.452, 0, 24.39, 72.485]
  MoveL 8198 to (10.76, -45.43, -10.97) mm, rotated rx -180 ry 0 rz 90 deg; joints [72.466, -16.85, 82.544, 0, 24.306, 72.466]
  MoveL 8199 to (9.31, -45.88, -11.37) mm, rotated rx -180 ry 0 rz 90 deg; joints [72.437, -16.854, 82.624, 0, 24.23, 72.437]
  MoveL 8200 to (8, -46.64, -11.78) mm, rotated rx 180 ry 0 rz 90 deg; joints [72.4, -16.854, 82.687, 0, 24.167, 72.4]
  MoveL 8201 to (6.88, -47.67, -12.19) mm, rotated rx 180 ry 0 rz 90 deg; joints [72.356, -16.849, 82.73, 0, 24.119, 72.356]
  MoveL 8202 to (6.02, -48.93, -12.59) mm, rotated rx 180 ry 0 rz 90 deg; joints [72.308, -16.837, 82.749, 0, 24.088, 72.308]
  MoveL 8203 to (5.49, -50.35, -13) mm, rotated rx -180 ry 0 rz 90 deg; joints [72.257, -16.818, 82.741, 0, 24.077, 72.257]
  MoveL 8204 to (1.12, -66.33, -13) mm, rotated rx -180 ry 0 rz 90 deg; joints [71.706, -16.802, 82.681, 0, 24.121, 71.706]
  MoveC 8205 to (1.96, -68.67, -13) mm, rotated rx -180 ry 0 rz 90 deg; joints [71.641, -16.771, 82.566, 0, 24.205, 71.641] to (4.26, -69.57, -13) mm, rotated rx 180 ry 0 rz 90 deg; joints [71.637, -16.721, 82.38, 0, 24.341, 71.637]
  MoveC 8206 to (13.4, -69.21, -13) mm, rotated rx -180 ry 0 rz 90 deg; joints [71.743, -16.545, 81.733, 0, 24.813, 71.743] to (22.53, -68.76, -13) mm, rotated rx -180 ry 0 rz 90 deg; joints [71.851, -16.366, 81.083, 0, 25.284, 71.851]
  MoveL 8207 to (22.53, -40.73, -13) mm, rotated rx -180 ry 0 rz 90 deg; joints [72.731, -16.545, 81.732, 0, 24.813, 72.731]
  MoveC 8208 to (22.14, -40.28, -13) mm, rotated rx 180 ry 0 rz 90 deg; joints [72.741, -16.556, 81.77, 0, 24.785, 72.741] to (21.71, -39.87, -13) mm, rotated rx -180 ry 0 rz 90 deg; joints [72.75, -16.567, 81.811, 0, 24.756, 72.75]
  MoveL 8209 to (14.5, -33.81, -13) mm, rotated rx 180 ry 0 rz 90 deg; joints [72.871, -16.744, 82.467, 0, 24.278, 72.871]
  MoveL 8210 to (14.31, -33.66, -13) mm, rotated rx 180 ry 0 rz 90 deg; joints [72.874, -16.749, 82.484, 0, 24.265, 72.874]
  MoveC 8211 to (12.01, -33.28, -13) mm, rotated rx -180 ry 0 rz 90 deg; joints [72.864, -16.796, 82.657, 0, 24.138, 72.864] to (9.95, -34.39, -13) mm, rotated rx -180 ry 0 rz 90 deg; joints [72.808, -16.828, 82.78, 0, 24.048, 72.808]
  MoveL 8212 to (9.84, -34.59, -13) mm, rotated rx 180 ry 0 rz 90 deg; joints [72.801, -16.829, 82.784, 0, 24.046, 72.801]
  MoveL 8213 to (9.54, -35.54, -13) mm, rotated rx 180 ry 0 rz 90 deg; joints [72.768, -16.83, 82.785, 0, 24.045, 72.768]
  MoveL 8214 to (5.49, -50.35, -13) mm, rotated rx -180 ry 0 rz 90 deg; joints [72.257, -16.818, 82.741, 0, 24.077, 72.257]
  MoveL 8215 to (12.77, -52.34, -13) mm, rotated rx 180 ry 0 rz 90 deg; joints [72.268, -16.665, 82.173, 0, 24.492, 72.268]
  MoveL 8216 to (12.77, -52.34, -10) mm, rotated rx 180 ry 0 rz 90 deg; joints [72.268, -16.817, 82.276, 0, 24.542, 72.268]
  Establecer velocidad (1000.0 mm/s)
  MoveL 8217 to (12.77, -52.34, 10) mm, rotated rx -180 ry 0 rz 90 deg; joints [72.268, -17.832, 82.948, 0, 24.884, 72.268]
  Establecer velocidad (66.7 mm/s)
  MoveL 8218 to (-38.89, -52.14, 10) mm, rotated rx 180 ry 0 rz 90 deg; joints [71.738, -18.794, 86.586, 0, 22.208, 71.738]
  MoveL 8219 to (-38.89, -52.14, -9.75) mm, rotated rx -180 ry 0 rz 90 deg; joints [71.738, -17.777, 85.924, 0, 21.853, 71.738]
  MoveL 8220 to (-37.48, -52.69, -10.16) mm, rotated rx -180 ry 0 rz 90 deg; joints [71.735, -17.729, 85.8, 0, 21.929, 71.735]
  MoveL 8221 to (-35.97, -52.89, -10.56) mm, rotated rx -180 ry 0 rz 90 deg; joints [71.745, -17.681, 85.678, 0, 22.003, 71.745]
  MoveL 8222 to (-34.46, -52.75, -10.97) mm, rotated rx 180 ry 0 rz 90 deg; joints [71.765, -17.635, 85.563, 0, 22.072, 71.765]
  MoveL 8223 to (-33.01, -52.28, -11.37) mm, rotated rx 180 ry 0 rz 90 deg; joints [71.796, -17.591, 85.459, 0, 22.132, 71.796]
  MoveL 8224 to (-31.71, -51.5, -11.78) mm, rotated rx 180 ry 0 rz 90 deg; joints [71.835, -17.552, 85.373, 0, 22.179, 71.835]
  MoveL 8225 to (-30.6, -50.45, -12.19) mm, rotated rx -180 ry 0 rz 90 deg; joints [71.88, -17.518, 85.307, 0, 22.212, 71.88]
  MoveL 8226 to (-29.77, -49.19, -12.59) mm, rotated rx 180 ry 0 rz 90 deg; joints [71.93, -17.49, 85.263, 0, 22.227, 71.93]
  MoveL 8227 to (-29.26, -47.76, -13) mm, rotated rx -180 ry 0 rz 90 deg; joints [71.981, -17.468, 85.246, 0, 22.222, 71.981]
  MoveL 8228 to (-24.17, -27.95, -13) mm, rotated rx -180 ry 0 rz 90 deg; joints [72.675, -17.49, 85.331, 0, 22.158, 72.675]
  MoveL 8229 to (-23.96, -27.13, -13) mm, rotated rx -180 ry 0 rz 90 deg; joints [72.703, -17.49, 85.335, 0, 22.156, 72.703]
  MoveC 8230 to (-23.9, -26.61, -13) mm, rotated rx -180 ry 0 rz 90 deg; joints [72.721, -17.492, 85.342, 0, 22.151, 72.721] to (-23.96, -26.08, -13) mm, rotated rx -180 ry 0 rz 90 deg; joints [72.737, -17.496, 85.357, 0, 22.139, 72.737]
  MoveC 8231 to (-24.89, -24.38, -13) mm, rotated rx -180 ry 0 rz 90 deg; joints [72.783, -17.522, 85.459, 0, 22.063, 72.783] to (-26.54, -23.35, -13) mm, rotated rx 180 ry 0 rz 90 deg; joints [72.8, -17.556, 85.595, 0, 21.96, 72.8]
  MoveL 8232 to (-26.8, -23.29, -13) mm, rotated rx 180 ry 0 rz 90 deg; joints [72.799, -17.56, 85.615, 0, 21.946, 72.799]
  MoveL 8233 to (-27.96, -23.47, -13) mm, rotated rx -180 ry 0 rz 90 deg; joints [72.782, -17.579, 85.691, 0, 21.888, 72.782]
  MoveC 8234 to (-48.57, -27.58, -13) mm, rotated rx -180 ry 0 rz 90 deg; joints [72.437, -17.904, 87.022, 0, 20.882, 72.437] to (-69.17, -31.76, -13) mm, rotated rx 180 ry 0 rz 90 deg; joints [72.081, -18.21, 88.326, 0, 19.884, 72.081]
  MoveC 8235 to (-70.7, -32.66, -13) mm, rotated rx -180 ry 0 rz 90 deg; joints [72.035, -18.229, 88.409, 0, 19.82, 72.035] to (-71.34, -34.32, -13) mm, rotated rx -180 ry 0 rz 90 deg; joints [71.973, -18.231, 88.416, 0, 19.815, 71.973]
  MoveL 8236 to (-71.36, -34.59, -13) mm, rotated rx -180 ry 0 rz 90 deg; joints [71.964, -18.23, 88.411, 0, 19.818, 71.964]
  MoveL 8237 to (-71.36, -68.26, -13) mm, rotated rx -180 ry 0 rz 90 deg; joints [70.855, -18.053, 87.651, 0, 20.402, 70.855]
  MoveC 8238 to (-70.52, -70.25, -13) mm, rotated rx 180 ry 0 rz 90 deg; joints [70.8, -18.029, 87.548, 0, 20.481, 70.8] to (-68.52, -71.06, -13) mm, rotated rx 180 ry 0 rz 90 deg; joints [70.796, -17.993, 87.395, 0, 20.598, 70.796]
  MoveC 8239 to (-52.9, -70.8, -13) mm, rotated rx -180 ry 0 rz 90 deg; joints [70.98, -17.74, 86.342, 0, 21.398, 70.98] to (-37.27, -70.49, -13) mm, rotated rx -180 ry 0 rz 90 deg; joints [71.163, -17.476, 85.277, 0, 22.199, 71.163]
  MoveC 8240 to (-35.57, -69.88, -13) mm, rotated rx 180 ry 0 rz 90 deg; joints [71.201, -17.45, 85.174, 0, 22.276, 71.201] to (-34.56, -68.38, -13) mm, rotated rx 180 ry 0 rz 90 deg; joints [71.261, -17.441, 85.139, 0, 22.302, 71.261]
  MoveL 8241 to (-34.39, -67.76, -13) mm, rotated rx 180 ry 0 rz 90 deg; joints [71.283, -17.442, 85.142, 0, 22.3, 71.283]
  MoveL 8242 to (-29.26, -47.76, -13) mm, rotated rx -180 ry 0 rz 90 deg; joints [71.981, -17.468, 85.246, 0, 22.222, 71.981]
  MoveL 8243 to (-36.57, -45.88, -13) mm, rotated rx -180 ry 0 rz 90 deg; joints [71.965, -17.605, 85.794, 0, 21.811, 71.965]
  MoveL 8244 to (-36.57, -45.88, -10) mm, rotated rx -180 ry 0 rz 90 deg; joints [71.965, -17.76, 85.897, 0, 21.863, 71.965]
  Establecer velocidad (1000.0 mm/s)
  MoveL 8245 to (-36.57, -45.88, 10) mm, rotated rx -180 ry 0 rz 90 deg; joints [71.965, -18.789, 86.567, 0, 22.222, 71.965]
  Establecer velocidad (66.7 mm/s)
  MoveL 8246 to (-39.03, -52.11, 10) mm, rotated rx 180 ry 0 rz 90 deg; joints [71.737, -18.796, 86.596, 0, 22.2, 71.737]
  MoveL 8247 to (-39.03, -52.11, -10) mm, rotated rx -180 ry 0 rz 90 deg; joints [71.737, -17.767, 85.926, 0, 21.841, 71.737]
  MoveL 8248 to (-37.62, -52.66, -10.41) mm, rotated rx 180 ry 0 rz 90 deg; joints [71.735, -17.719, 85.802, 0, 21.916, 71.735]
  MoveL 8249 to (-36.11, -52.85, -10.81) mm, rotated rx 180 ry 0 rz 90 deg; joints [71.744, -17.671, 85.68, 0, 21.991, 71.744]
  MoveL 8250 to (-34.6, -52.72, -11.22) mm, rotated rx 180 ry 0 rz 90 deg; joints [71.765, -17.624, 85.565, 0, 22.06, 71.765]
  MoveL 8251 to (-33.15, -52.24, -11.63) mm, rotated rx 180 ry 0 rz 90 deg; joints [71.795, -17.581, 85.462, 0, 22.119, 71.795]
  MoveL 8252 to (-31.85, -51.47, -12.03) mm, rotated rx -180 ry 0 rz 90 deg; joints [71.834, -17.542, 85.375, 0, 22.167, 71.834]
  MoveL 8253 to (-30.75, -50.42, -12.44) mm, rotated rx -180 ry 0 rz 90 deg; joints [71.88, -17.508, 85.309, 0, 22.199, 71.88]
  MoveL 8254 to (-29.91, -49.15, -12.84) mm, rotated rx 180 ry 0 rz 90 deg; joints [71.93, -17.48, 85.266, 0, 22.214, 71.93]
  MoveL 8255 to (-29.4, -47.72, -13.25) mm, rotated rx 180 ry 0 rz 90 deg; joints [71.981, -17.458, 85.248, 0, 22.21, 71.981]
  MoveL 8256 to (-24.17, -27.32, -13.25) mm, rotated rx -180 ry 0 rz 90 deg; joints [72.695, -17.48, 85.336, 0, 22.144, 72.695]
  MoveL 8257 to (-24.09, -27.01, -13.25) mm, rotated rx 180 ry 0 rz 90 deg; joints [72.706, -17.48, 85.338, 0, 22.142, 72.706]
  MoveC 8258 to (-24.5, -25.41, -13.25) mm, rotated rx -180 ry 0 rz 90 deg; joints [72.754, -17.496, 85.401, 0, 22.095, 72.754] to (-25.58, -24.17, -13.25) mm, rotated rx -180 ry 0 rz 90 deg; joints [72.783, -17.522, 85.503, 0, 22.019, 72.783]
  MoveL 8259 to (-26, -23.87, -13.25) mm, rotated rx 180 ry 0 rz 90 deg; joints [72.789, -17.531, 85.538, 0, 21.992, 72.789]
  MoveC 8260 to (-26.71, -23.56, -13.25) mm, rotated rx -180 ry 0 rz 90 deg; joints [72.791, -17.545, 85.595, 0, 21.95, 72.791] to (-27.49, -23.56, -13.25) mm, rotated rx 180 ry 0 rz 90 deg; joints [72.784, -17.558, 85.649, 0, 21.909, 72.784]
  MoveC 8261 to (-48.27, -27.68, -13.25) mm, rotated rx -180 ry 0 rz 90 deg; joints [72.436, -17.885, 86.99, 0, 20.895, 72.436] to (-69.03, -31.88, -13.25) mm, rotated rx -180 ry 0 rz 90 deg; joints [72.079, -18.194, 88.305, 0, 19.889, 72.079]
  MoveC 8262 to (-70.55, -32.79, -13.25) mm, rotated rx -180 ry 0 rz 90 deg; joints [72.032, -18.213, 88.388, 0, 19.826, 72.032] to (-71.17, -34.44, -13.25) mm, rotated rx 180 ry 0 rz 90 deg; joints [71.971, -18.214, 88.393, 0, 19.821, 71.971]
  MoveL 8263 to (-71.19, -35.54, -13.25) mm, rotated rx 180 ry 0 rz 90 deg; joints [71.934, -18.209, 88.371, 0, 19.838, 71.934]
  MoveL 8264 to (-71.19, -68.19, -13.25) mm, rotated rx 180 ry 0 rz 90 deg; joints [70.86, -18.038, 87.633, 0, 20.405, 70.86]
  MoveC 8265 to (-70.4, -70.1, -13.25) mm, rotated rx 180 ry 0 rz 90 deg; joints [70.806, -18.015, 87.535, 0, 20.48, 70.806] to (-68.5, -70.9, -13.25) mm, rotated rx 180 ry 0 rz 90 deg; joints [70.801, -17.98, 87.388, 0, 20.592, 70.801]
  MoveL 8266 to (-67.76, -70.91, -13.25) mm, rotated rx -180 ry 0 rz 90 deg; joints [70.81, -17.968, 87.338, 0, 20.63, 70.81]
  MoveL 8267 to (-63.99, -70.85, -13.25) mm, rotated rx 180 ry 0 rz 90 deg; joints [70.854, -17.908, 87.085, 0, 20.823, 70.854]
  MoveC 8268 to (-50.67, -70.61, -13.25) mm, rotated rx 180 ry 0 rz 90 deg; joints [71.012, -17.691, 86.186, 0, 21.505, 71.012] to (-37.35, -70.32, -13.25) mm, rotated rx -180 ry 0 rz 90 deg; joints [71.168, -17.465, 85.278, 0, 22.188, 71.168]
  MoveC 8269 to (-35.65, -69.71, -13.25) mm, rotated rx 180 ry 0 rz 90 deg; joints [71.206, -17.439, 85.174, 0, 22.265, 71.206] to (-34.66, -68.19, -13.25) mm, rotated rx -180 ry 0 rz 90 deg; joints [71.266, -17.431, 85.142, 0, 22.289, 71.266]
  MoveL 8270 to (-33.57, -63.97, -13.25) mm, rotated rx 180 ry 0 rz 90 deg; joints [71.413, -17.437, 85.165, 0, 22.272, 71.413]
  MoveL 8271 to (-29.4, -47.72, -13.25) mm, rotated rx 180 ry 0 rz 90 deg; joints [71.981, -17.458, 85.248, 0, 22.21, 71.981]
  MoveL 8272 to (-36.71, -45.84, -13.25) mm, rotated rx 180 ry 0 rz 90 deg; joints [71.965, -17.595, 85.797, 0, 21.798, 71.965]
  MoveL 8273 to (-36.71, -45.84, -10.25) mm, rotated rx 180 ry 0 rz 90 deg; joints [71.965, -17.75, 85.899, 0, 21.85, 71.965]
  Establecer velocidad (1000.0 mm/s)
  MoveL 8274 to (-36.71, -45.84, 10) mm, rotated rx -180 ry 0 rz 90 deg; joints [71.965, -18.792, 86.578, 0, 22.214, 71.965]
  Establecer velocidad (66.7 mm/s)
  MoveL 8275 to (15.29, -46.58, 10) mm, rotated rx 180 ry 0 rz 90 deg; joints [72.475, -17.818, 82.898, 0, 24.92, 72.475]
  MoveL 8276 to (15.29, -46.58, -10) mm, rotated rx 180 ry 0 rz 90 deg; joints [72.475, -16.804, 82.226, 0, 24.578, 72.475]
  MoveL 8277 to (13.89, -46, -10.41) mm, rotated rx 180 ry 0 rz 90 deg; joints [72.479, -16.814, 82.326, 0, 24.488, 72.479]
  MoveL 8278 to (12.39, -45.78, -10.81) mm, rotated rx 180 ry 0 rz 90 deg; joints [72.471, -16.824, 82.425, 0, 24.399, 72.471]
  MoveL 8279 to (10.87, -45.89, -11.22) mm, rotated rx -180 ry 0 rz 90 deg; joints [72.452, -16.832, 82.517, 0, 24.315, 72.452]
  MoveL 8280 to (9.42, -46.34, -11.63) mm, rotated rx -180 ry 0 rz 90 deg; joints [72.424, -16.837, 82.597, 0, 24.239, 72.424]
  MoveL 8281 to (8.1, -47.1, -12.03) mm, rotated rx 180 ry 0 rz 90 deg; joints [72.386, -16.837, 82.661, 0, 24.176, 72.386]
  MoveL 8282 to (6.98, -48.13, -12.44) mm, rotated rx 180 ry 0 rz 90 deg; joints [72.343, -16.831, 82.703, 0, 24.128, 72.343]
  MoveL 8283 to (6.12, -49.38, -12.84) mm, rotated rx 180 ry 0 rz 90 deg; joints [72.294, -16.819, 82.722, 0, 24.097, 72.294]
  MoveL 8284 to (5.59, -50.8, -13.25) mm, rotated rx -180 ry 0 rz 90 deg; joints [72.244, -16.8, 82.714, 0, 24.086, 72.244]
  MoveL 8285 to (1.46, -65.86, -13.25) mm, rotated rx -180 ry 0 rz 90 deg; joints [71.725, -16.786, 82.66, 0, 24.126, 71.725]
  MoveL 8286 to (1.35, -66.33, -13.25) mm, rotated rx 180 ry 0 rz 90 deg; joints [71.709, -16.785, 82.656, 0, 24.129, 71.709]
  MoveC 8287 to (2.26, -68.52, -13.25) mm, rotated rx -180 ry 0 rz 90 deg; joints [71.649, -16.753, 82.539, 0, 24.214, 71.649] to (4.47, -69.37, -13.25) mm, rotated rx -180 ry 0 rz 90 deg; joints [71.646, -16.706, 82.362, 0, 24.344, 71.646]
  MoveC 8288 to (12.07, -69.06, -13.25) mm, rotated rx 180 ry 0 rz 90 deg; joints [71.734, -16.56, 81.823, 0, 24.736, 71.734] to (19.67, -68.67, -13.25) mm, rotated rx -180 ry 0 rz 90 deg; joints [71.825, -16.411, 81.283, 0, 25.128, 71.825]
  MoveL 8289 to (19.67, -38.45, -13.25) mm, rotated rx -180 ry 0 rz 90 deg; joints [72.775, -16.603, 81.982, 0, 24.621, 72.775]
  MoveL 8290 to (14.5, -34.07, -13.25) mm, rotated rx -180 ry 0 rz 90 deg; joints [72.863, -16.73, 82.452, 0, 24.278, 72.863]
  MoveC 8291 to (12.45, -33.61, -13.25) mm, rotated rx 180 ry 0 rz 90 deg; joints [72.857, -16.772, 82.609, 0, 24.163, 72.857] to (10.49, -34.34, -13.25) mm, rotated rx 180 ry 0 rz 90 deg; joints [72.815, -16.806, 82.734, 0, 24.071, 72.815]
  MoveC 8292 to (10.09, -34.75, -13.25) mm, rotated rx -180 ry 0 rz 90 deg; joints [72.798, -16.811, 82.754, 0, 24.057, 72.798] to (9.85, -35.27, -13.25) mm, rotated rx 180 ry 0 rz 90 deg; joints [72.779, -16.812, 82.759, 0, 24.053, 72.779]
  MoveL 8293 to (5.59, -50.8, -13.25) mm, rotated rx -180 ry 0 rz 90 deg; joints [72.244, -16.8, 82.714, 0, 24.086, 72.244]
  MoveL 8294 to (12.87, -52.8, -13.25) mm, rotated rx -180 ry 0 rz 90 deg; joints [72.254, -16.647, 82.146, 0, 24.501, 72.254]
  MoveL 8295 to (12.12, -55.52, -13.25) mm, rotated rx -180 ry 0 rz 90 deg; joints [72.161, -16.645, 82.137, 0, 24.508, 72.161]
  MoveL 8296 to (12.12, -55.52, -10.25) mm, rotated rx -180 ry 0 rz 90 deg; joints [72.161, -16.797, 82.24, 0, 24.557, 72.161]
  Establecer velocidad (1000.0 mm/s)
  MoveL 8297 to (12.12, -55.52, 10) mm, rotated rx -180 ry 0 rz 90 deg; joints [72.161, -17.824, 82.921, 0, 24.904, 72.161]
  Establecer velocidad (66.7 mm/s)
  MoveL 8298 to (16.34, 13.31, 10) mm, rotated rx 180 ry 0 rz 90 deg; joints [74.395, -18.146, 84.103, 0, 24.043, 74.395]
  MoveL 8299 to (16.34, 13.31, -10) mm, rotated rx 180 ry 0 rz 90 deg; joints [74.395, -17.127, 83.431, 0, 23.696, 74.395]
  MoveL 8300 to (16.54, 12.79, -10.15) mm, rotated rx 180 ry 0 rz 90 deg; joints [74.38, -17.113, 83.402, 0, 23.711, 74.38]
  MoveL 8301 to (16.9, 11.93, -10.4) mm, rotated rx 180 ry 0 rz 90 deg; joints [74.355, -17.089, 83.35, 0, 23.739, 74.355]
  MoveL 8302 to (17.21, 11.53, -10.53) mm, rotated rx 180 ry 0 rz 90 deg; joints [74.345, -17.074, 83.315, 0, 23.759, 74.345]
  MoveL 8303 to (19.67, 9.72, -11.35) mm, rotated rx -180 ry 0 rz 90 deg; joints [74.309, -16.975, 83.074, 0, 23.902, 74.309]
  MoveL 8304 to (19.67, 16.8, -13.25) mm, rotated rx -180 ry 0 rz 90 deg; joints [74.537, -16.916, 83.151, 0, 23.766, 74.537]
  MoveL 8305 to (19.67, 23.88, -13.25) mm, rotated rx 180 ry 0 rz 90 deg; joints [74.765, -16.953, 83.29, 0, 23.663, 74.765]
  MoveL 8306 to (16.58, 23.91, -13.25) mm, rotated rx -180 ry 0 rz 90 deg; joints [74.739, -17.012, 83.513, 0, 23.499, 74.739]
  MoveC 8307 to (14.46, 22.99, -13.25) mm, rotated rx 180 ry 0 rz 90 deg; joints [74.69, -17.047, 83.647, 0, 23.4, 74.69] to (13.59, 20.85, -13.25) mm, rotated rx 180 ry 0 rz 90 deg; joints [74.613, -17.052, 83.667, 0, 23.385, 74.613]
  MoveC 8308 to (13.63, 20.61, -13.25) mm, rotated rx 180 ry 0 rz 90 deg; joints [74.606, -17.05, 83.66, 0, 23.39, 74.606] to (13.7, 20.38, -13.25) mm, rotated rx 180 ry 0 rz 90 deg; joints [74.599, -17.048, 83.651, 0, 23.397, 74.599]
  MoveL 8309 to (16.54, 12.79, -13.25) mm, rotated rx 180 ry 0 rz 90 deg; joints [74.38, -16.955, 83.296, 0, 23.659, 74.38]
  MoveL 8310 to (16.75, 12.27, -13.25) mm, rotated rx -180 ry 0 rz 90 deg; joints [74.365, -16.948, 83.27, 0, 23.678, 74.365]
  MoveC 8311 to (17.07, 11.74, -13.25) mm, rotated rx 180 ry 0 rz 90 deg; joints [74.351, -16.939, 83.237, 0, 23.702, 74.351] to (17.51, 11.31, -13.25) mm, rotated rx 180 ry 0 rz 90 deg; joints [74.341, -16.928, 83.196, 0, 23.732, 74.341]
  MoveL 8312 to (19.67, 9.72, -13.25) mm, rotated rx -180 ry 0 rz 90 deg; joints [74.309, -16.879, 83.008, 0, 23.87, 74.309]
  MoveL 8313 to (19.67, 16.8, -13.25) mm, rotated rx -180 ry 0 rz 90 deg; joints [74.537, -16.916, 83.151, 0, 23.766, 74.537]
  MoveL 8314 to (15.9, 16.8, -13.25) mm, rotated rx 180 ry 0 rz 90 deg; joints [74.503, -16.988, 83.422, 0, 23.566, 74.503]
  MoveL 8315 to (15.9, 16.8, -10.25) mm, rotated rx 180 ry 0 rz 90 deg; joints [74.503, -17.141, 83.525, 0, 23.617, 74.503]
  Establecer velocidad (1000.0 mm/s)
  MoveL 8316 to (15.9, 16.8, 10) mm, rotated rx -180 ry 0 rz 90 deg; joints [74.503, -18.173, 84.204, 0, 23.969, 74.503]
  Establecer velocidad (66.7 mm/s)
  MoveL 8317 to (-6.36, 59.81, 10) mm, rotated rx 180 ry 0 rz 90 deg; joints [75.714, -18.796, 86.596, 0, 22.2, 75.714]
  MoveL 8318 to (-6.36, 59.81, -10) mm, rotated rx -180 ry 0 rz 90 deg; joints [75.714, -17.767, 85.926, 0, 21.841, 75.714]
  MoveL 8319 to (-5.15, 58.89, -10.41) mm, rotated rx -180 ry 0 rz 90 deg; joints [75.694, -17.721, 85.811, 0, 21.91, 75.694]
  MoveL 8320 to (-3.73, 58.36, -10.81) mm, rotated rx -180 ry 0 rz 90 deg; joints [75.688, -17.672, 85.687, 0, 21.985, 75.688]
  MoveL 8321 to (-2.21, 58.23, -11.22) mm, rotated rx 180 ry 0 rz 90 deg; joints [75.697, -17.624, 85.564, 0, 22.06, 75.697]
  MoveL 8322 to (-0.72, 58.51, -11.63) mm, rotated rx -180 ry 0 rz 90 deg; joints [75.718, -17.578, 85.45, 0, 22.128, 75.718]
  MoveL 8323 to (0.65, 59.18, -12.03) mm, rotated rx 180 ry 0 rz 90 deg; joints [75.752, -17.536, 85.352, 0, 22.184, 75.752]
  MoveL 8324 to (1.78, 60.2, -12.44) mm, rotated rx -180 ry 0 rz 90 deg; joints [75.795, -17.5, 85.276, 0, 22.224, 75.795]
  MoveL 8325 to (2.6, 61.48, -12.84) mm, rotated rx -180 ry 0 rz 90 deg; joints [75.844, -17.47, 85.227, 0, 22.243, 75.844]
  MoveL 8326 to (3.02, 62.93, -13.25) mm, rotated rx 180 ry 0 rz 90 deg; joints [75.895, -17.448, 85.209, 0, 22.239, 75.895]
  MoveL 8327 to (4.05, 69.18, -13.25) mm, rotated rx 180 ry 0 rz 90 deg; joints [76.109, -17.457, 85.246, 0, 22.211, 76.109]
  MoveC 8328 to (-3.76, 69.48, -13.25) mm, rotated rx -180 ry 0 rz 90 deg; joints [76.055, -17.596, 85.803, 0, 21.793, 76.055] to (-11.58, 69.75, -13.25) mm, rotated rx -180 ry 0 rz 90 deg; joints [76, -17.732, 86.357, 0, 21.376, 76]
  MoveC 8329 to (-13.61, 67.28, -13.25) mm, rotated rx 180 ry 0 rz 90 deg; joints [75.901, -17.756, 86.455, 0, 21.301, 75.901] to (-13.4, 64.08, -13.25) mm, rotated rx 180 ry 0 rz 90 deg; joints [75.796, -17.739, 86.385, 0, 21.355, 75.796]
  MoveL 8330 to (-7.11, 59.94, -13.25) mm, rotated rx 180 ry 0 rz 90 deg; joints [75.712, -17.613, 85.87, 0, 21.743, 75.712]
  MoveL 8331 to (-6.16, 59.3, -13.25) mm, rotated rx -180 ry 0 rz 90 deg; joints [75.699, -17.594, 85.792, 0, 21.802, 75.699]
  MoveL 8332 to (-4.99, 58.48, -13.25) mm, rotated rx 180 ry 0 rz 90 deg; joints [75.681, -17.569, 85.695, 0, 21.875, 75.681]
  MoveC 8333 to (-4.63, 58.25, -13.25) mm, rotated rx 180 ry 0 rz 90 deg; joints [75.677, -17.562, 85.666, 0, 21.897, 75.677] to (-4.26, 58.06, -13.25) mm, rotated rx 180 ry 0 rz 90 deg; joints [75.674, -17.555, 85.636, 0, 21.919, 75.674]
  MoveC 8334 to (7.71, 59.29, -13.25) mm, rotated rx 180 ry 0 rz 90 deg; joints [75.814, -17.347, 84.811, 0, 22.536, 75.814] to (19.67, 60.72, -13.25) mm, rotated rx -180 ry 0 rz 90 deg; joints [75.959, -17.134, 83.982, 0, 23.152, 75.959]
  MoveL 8335 to (19.67, 68.51, -13.25) mm, rotated rx -180 ry 0 rz 90 deg; joints [76.213, -17.17, 84.121, 0, 23.05, 76.213]
  MoveC 8336 to (11.86, 68.86, -13.25) mm, rotated rx -180 ry 0 rz 90 deg; joints [76.162, -17.315, 84.685, 0, 22.63, 76.162] to (4.05, 69.18, -13.25) mm, rotated rx 180 ry 0 rz 90 deg; joints [76.109, -17.457, 85.246, 0, 22.211, 76.109]
  MoveL 8337 to (3.75, 61.64, -13.25) mm, rotated rx 180 ry 0 rz 90 deg; joints [75.859, -17.429, 85.134, 0, 22.295, 75.859]
  MoveL 8338 to (3.75, 61.64, -10.25) mm, rotated rx -180 ry 0 rz 90 deg; joints [75.859, -17.584, 85.237, 0, 22.347, 75.859]
  Establecer velocidad (1000.0 mm/s)
  MoveL 8339 to (3.75, 61.64, 10) mm, rotated rx 180 ry 0 rz 90 deg; joints [75.859, -18.623, 85.916, 0, 22.707, 75.859]
  Establecer velocidad (66.7 mm/s)
  MoveL 8340 to (-62.95, 35.42, 10) mm, rotated rx 180 ry 0 rz 90 deg; joints [74.393, -19.626, 90.042, 0, 19.584, 74.393]
  MoveL 8341 to (-62.95, 35.42, -10) mm, rotated rx 180 ry 0 rz 90 deg; joints [74.393, -18.581, 89.372, 0, 19.209, 74.393]
  MoveL 8342 to (-64.46, 35.61, -10.41) mm, rotated rx 180 ry 0 rz 90 deg; joints [74.385, -18.583, 89.463, 0, 19.12, 74.385]
  MoveL 8343 to (-65.97, 35.42, -10.81) mm, rotated rx 180 ry 0 rz 90 deg; joints [74.365, -18.583, 89.547, 0, 19.036, 74.365]
  MoveL 8344 to (-67.4, 34.91, -11.22) mm, rotated rx 180 ry 0 rz 90 deg; joints [74.334, -18.581, 89.62, 0, 18.962, 74.334]
  MoveL 8345 to (-68.68, 34.09, -11.63) mm, rotated rx 180 ry 0 rz 90 deg; joints [74.294, -18.575, 89.676, 0, 18.899, 74.294]
  MoveL 8346 to (-69.75, 33.01, -12.03) mm, rotated rx 180 ry 0 rz 90 deg; joints [74.247, -18.565, 89.714, 0, 18.852, 74.247]
  MoveL 8347 to (-70.56, 31.73, -12.44) mm, rotated rx 180 ry 0 rz 90 deg; joints [74.196, -18.551, 89.729, 0, 18.821, 74.196]
  MoveL 8348 to (-71.05, 30.29, -12.84) mm, rotated rx 180 ry 0 rz 90 deg; joints [74.143, -18.531, 89.722, 0, 18.809, 74.143]
  MoveL 8349 to (-71.19, 28.78, -13.25) mm, rotated rx 180 ry 0 rz 90 deg; joints [74.09, -18.505, 89.688, 0, 18.817, 74.09]
  MoveL 8350 to (-71.19, 4.26, -13.25) mm, rotated rx 180 ry 0 rz 90 deg; joints [73.262, -18.399, 89.207, 0, 19.191, 73.262]
  MoveL 8351 to (-71.18, 3.79, -13.25) mm, rotated rx 180 ry 0 rz 90 deg; joints [73.247, -18.396, 89.197, 0, 19.199, 73.247]
  MoveC 8352 to (-70, 1.83, -13.25) mm, rotated rx 180 ry 0 rz 90 deg; joints [73.193, -18.37, 89.078, 0, 19.292, 73.193] to (-67.76, 1.39, -13.25) mm, rotated rx 180 ry 0 rz 90 deg; joints [73.201, -18.334, 88.919, 0, 19.415, 73.201]
  MoveC 8353 to (-46.42, 6.51, -13.25) mm, rotated rx -180 ry 0 rz 90 deg; joints [73.584, -18.025, 87.577, 0, 20.448, 73.584] to (-25.11, 11.73, -13.25) mm, rotated rx 180 ry 0 rz 90 deg; joints [73.961, -17.698, 86.215, 0, 21.483, 73.961]
  MoveC 8354 to (-24.27, 12.12, -13.25) mm, rotated rx 180 ry 0 rz 90 deg; joints [73.982, -17.685, 86.164, 0, 21.521, 73.982] to (-23.63, 12.79, -13.25) mm, rotated rx 180 ry 0 rz 90 deg; joints [74.01, -17.678, 86.133, 0, 21.544, 74.01]
  MoveC 8355 to (-23.03, 14.15, -13.25) mm, rotated rx 180 ry 0 rz 90 deg; joints [74.06, -17.674, 86.119, 0, 21.555, 74.06] to (-23.15, 15.64, -13.25) mm, rotated rx 180 ry 0 rz 90 deg; joints [74.108, -17.683, 86.156, 0, 21.527, 74.108]
  MoveL 8356 to (-27.96, 29.26, -13.25) mm, rotated rx -180 ry 0 rz 90 deg; joints [74.513, -17.829, 86.755, 0, 21.074, 74.513]
  MoveL 8357 to (-28.17, 29.85, -13.25) mm, rotated rx -180 ry 0 rz 90 deg; joints [74.531, -17.835, 86.781, 0, 21.054, 74.531]
  MoveC 8358 to (-28.56, 30.62, -13.25) mm, rotated rx -180 ry 0 rz 90 deg; joints [74.553, -17.845, 86.823, 0, 21.022, 74.553] to (-29.12, 31.27, -13.25) mm, rotated rx -180 ry 0 rz 90 deg; joints [74.569, -17.858, 86.874, 0, 20.984, 74.569]
  MoveL 8359 to (-29.79, 31.75, -13.25) mm, rotated rx 180 ry 0 rz 90 deg; joints [74.579, -17.871, 86.93, 0, 20.941, 74.579]
  MoveL 8360 to (-45.96, 42.39, -13.25) mm, rotated rx 180 ry 0 rz 90 deg; joints [74.786, -18.179, 88.24, 0, 19.94, 74.786]
  MoveL 8361 to (-49.75, 44.86, -13.25) mm, rotated rx -180 ry 0 rz 90 deg; joints [74.835, -18.249, 88.543, 0, 19.705, 74.835]
  MoveL 8362 to (-66.94, 56.09, -13.25) mm, rotated rx 180 ry 0 rz 90 deg; joints [75.058, -18.553, 89.908, 0, 18.645, 75.058]
  MoveC 8363 to (-67.34, 56.27, -13.25) mm, rotated rx 180 ry 0 rz 90 deg; joints [75.061, -18.56, 89.938, 0, 18.622, 75.061] to (-67.76, 56.35, -13.25) mm, rotated rx 180 ry 0 rz 90 deg; joints [75.06, -18.566, 89.968, 0, 18.598, 75.06]
  MoveC 8364 to (-69.47, 56.02, -13.25) mm, rotated rx 180 ry 0 rz 90 deg; joints [75.033, -18.59, 90.077, 0, 18.513, 75.033] to (-70.82, 54.91, -13.25) mm, rotated rx -180 ry 0 rz 90 deg; joints [74.983, -18.605, 90.147, 0, 18.458, 74.983]
  MoveC 8365 to (-71.1, 54.37, -13.25) mm, rotated rx 180 ry 0 rz 90 deg; joints [74.962, -18.607, 90.156, 0, 18.451, 74.962] to (-71.19, 53.77, -13.25) mm, rotated rx 180 ry 0 rz 90 deg; joints [74.941, -18.606, 90.151, 0, 18.454, 74.941]
  MoveL 8366 to (-71.19, 28.78, -13.25) mm, rotated rx 180 ry 0 rz 90 deg; joints [74.09, -18.505, 89.688, 0, 18.817, 74.09]
  MoveL 8367 to (-63.64, 28.78, -13.25) mm, rotated rx 180 ry 0 rz 90 deg; joints [74.163, -18.393, 89.181, 0, 19.211, 74.163]
  MoveL 8368 to (-63.64, 28.78, -10.25) mm, rotated rx 180 ry 0 rz 90 deg; joints [74.163, -18.55, 89.284, 0, 19.266, 74.163]
  Establecer velocidad (1000.0 mm/s)
  MoveL 8369 to (-63.64, 28.78, 10) mm, rotated rx 180 ry 0 rz 90 deg; joints [74.163, -19.608, 89.963, 0, 19.645, 74.163]
  Establecer velocidad (66.7 mm/s)
  MoveL 8370 to (-62.79, 35.42, 10) mm, rotated rx 180 ry 0 rz 90 deg; joints [74.395, -19.624, 90.031, 0, 19.592, 74.395]
  MoveL 8371 to (-62.79, 35.42, -10.25) mm, rotated rx -180 ry 0 rz 90 deg; joints [74.395, -18.565, 89.352, 0, 19.213, 74.395]
  MoveL 8372 to (-64.3, 35.61, -10.66) mm, rotated rx 180 ry 0 rz 90 deg; joints [74.387, -18.567, 89.443, 0, 19.124, 74.387]
  MoveL 8373 to (-65.8, 35.42, -11.06) mm, rotated rx -180 ry 0 rz 90 deg; joints [74.367, -18.568, 89.527, 0, 19.04, 74.367]
  MoveL 8374 to (-67.23, 34.91, -11.47) mm, rotated rx -180 ry 0 rz 90 deg; joints [74.336, -18.566, 89.6, 0, 18.966, 74.336]
  MoveL 8375 to (-68.52, 34.09, -11.87) mm, rotated rx -180 ry 0 rz 90 deg; joints [74.296, -18.56, 89.657, 0, 18.903, 74.296]
  MoveL 8376 to (-69.59, 33.01, -12.28) mm, rotated rx -180 ry 0 rz 90 deg; joints [74.249, -18.55, 89.694, 0, 18.856, 74.249]
  MoveL 8377 to (-70.39, 31.73, -12.69) mm, rotated rx 180 ry 0 rz 90 deg; joints [74.198, -18.535, 89.71, 0, 18.825, 74.198]
  MoveL 8378 to (-70.89, 30.29, -13.09) mm, rotated rx -180 ry 0 rz 90 deg; joints [74.144, -18.515, 89.702, 0, 18.813, 74.144]
  MoveL 8379 to (-71.03, 28.78, -13.5) mm, rotated rx 180 ry 0 rz 90 deg; joints [74.092, -18.49, 89.669, 0, 18.821, 74.092]
  MoveL 8380 to (-71.03, 4.26, -13.5) mm, rotated rx 180 ry 0 rz 90 deg; joints [73.264, -18.383, 89.188, 0, 19.195, 73.264]
  MoveC 8381 to (-70.36, 2.48, -13.5) mm, rotated rx 180 ry 0 rz 90 deg; joints [73.211, -18.365, 89.107, 0, 19.258, 73.211] to (-68.7, 1.52, -13.5) mm, rotated rx 180 ry 0 rz 90 deg; joints [73.196, -18.336, 88.977, 0, 19.359, 73.196]
  MoveL 8382 to (-68.23, 1.47, -13.5) mm, rotated rx 180 ry 0 rz 90 deg; joints [73.199, -18.328, 88.944, 0, 19.385, 73.199]
  MoveL 8383 to (-67.76, 1.54, -13.5) mm, rotated rx -180 ry 0 rz 90 deg; joints [73.206, -18.322, 88.913, 0, 19.408, 73.206]
  MoveL 8384 to (-67.28, 1.65, -13.5) mm, rotated rx 180 ry 0 rz 90 deg; joints [73.214, -18.315, 88.884, 0, 19.431, 73.214]
  MoveC 8385 to (-46.18, 6.72, -13.5) mm, rotated rx 180 ry 0 rz 90 deg; joints [73.593, -18.009, 87.557, 0, 20.452, 73.593] to (-25.11, 11.91, -13.5) mm, rotated rx 180 ry 0 rz 90 deg; joints [73.967, -17.686, 86.21, 0, 21.476, 73.967]
  MoveC 8386 to (-23.83, 12.9, -13.5) mm, rotated rx -180 ry 0 rz 90 deg; joints [74.012, -17.669, 86.14, 0, 21.528, 74.012] to (-23.22, 14.4, -13.5) mm, rotated rx 180 ry 0 rz 90 deg; joints [74.067, -17.666, 86.128, 0, 21.538, 74.067]
  MoveL 8387 to (-23.18, 14.69, -13.5) mm, rotated rx -180 ry 0 rz 90 deg; joints [74.077, -17.666, 86.131, 0, 21.535, 74.077]
  MoveC 8388 to (-23.19, 15.17, -13.5) mm, rotated rx 180 ry 0 rz 90 deg; joints [74.092, -17.669, 86.142, 0, 21.527, 74.092] to (-23.32, 15.64, -13.5) mm, rotated rx 180 ry 0 rz 90 deg; joints [74.106, -17.674, 86.16, 0, 21.514, 74.106]
  MoveL 8389 to (-23.65, 16.58, -13.5) mm, rotated rx 180 ry 0 rz 90 deg; joints [74.135, -17.684, 86.201, 0, 21.482, 74.135]
  MoveL 8390 to (-28.22, 29.55, -13.5) mm, rotated rx 180 ry 0 rz 90 deg; joints [74.52, -17.822, 86.77, 0, 21.051, 74.52]
  MoveC 8391 to (-28.5, 30.19, -13.5) mm, rotated rx 180 ry 0 rz 90 deg; joints [74.539, -17.83, 86.802, 0, 21.027, 74.539] to (-28.86, 30.8, -13.5) mm, rotated rx 180 ry 0 rz 90 deg; joints [74.556, -17.838, 86.839, 0, 21, 74.556]
  MoveC 8392 to (-29.19, 31.12, -13.5) mm, rotated rx 180 ry 0 rz 90 deg; joints [74.563, -17.845, 86.868, 0, 20.978, 74.563] to (-29.56, 31.4, -13.5) mm, rotated rx 180 ry 0 rz 90 deg; joints [74.569, -17.853, 86.899, 0, 20.954, 74.569]
  MoveC 8393 to (-48.16, 43.66, -13.5) mm, rotated rx 180 ry 0 rz 90 deg; joints [74.809, -18.206, 88.404, 0, 19.802, 74.809] to (-66.81, 55.83, -13.5) mm, rotated rx 180 ry 0 rz 90 deg; joints [75.051, -18.537, 89.886, 0, 18.651, 75.051]
  MoveL 8394 to (-67.28, 56.04, -13.5) mm, rotated rx 180 ry 0 rz 90 deg; joints [75.054, -18.545, 89.922, 0, 18.623, 75.054]
  MoveC 8395 to (-69.5, 55.69, -13.5) mm, rotated rx 180 ry 0 rz 90 deg; joints [75.022, -18.576, 90.064, 0, 18.511, 75.022] to (-71, 54.01, -13.5) mm, rotated rx -180 ry 0 rz 90 deg; joints [74.95, -18.591, 90.134, 0, 18.457, 74.95]
  MoveC 8396 to (-71.02, 53.76, -13.5) mm, rotated rx 180 ry 0 rz 90 deg; joints [74.942, -18.59, 90.131, 0, 18.459, 74.942] to (-71.03, 53.52, -13.5) mm, rotated rx 180 ry 0 rz 90 deg; joints [74.933, -18.589, 90.127, 0, 18.462, 74.933]
  MoveL 8397 to (-71.03, 28.78, -13.5) mm, rotated rx 180 ry 0 rz 90 deg; joints [74.092, -18.49, 89.669, 0, 18.821, 74.092]
  MoveL 8398 to (-63.48, 28.78, -13.5) mm, rotated rx -180 ry 0 rz 90 deg; joints [74.164, -18.377, 89.162, 0, 19.216, 74.164]
  MoveL 8399 to (-63.48, 28.78, -10.5) mm, rotated rx 180 ry 0 rz 90 deg; joints [74.164, -18.534, 89.264, 0, 19.27, 74.164]
  Establecer velocidad (1000.0 mm/s)
  MoveL 8400 to (-63.48, 28.78, 10) mm, rotated rx 180 ry 0 rz 90 deg; joints [74.164, -19.605, 89.952, 0, 19.654, 74.164]
  Establecer velocidad (66.7 mm/s)
  MoveL 8401 to (-5.86, 59.5, 10) mm, rotated rx -180 ry 0 rz 90 deg; joints [75.708, -18.786, 86.556, 0, 22.23, 75.708]
  MoveL 8402 to (-5.86, 59.5, -10.25) mm, rotated rx -180 ry 0 rz 90 deg; joints [75.708, -17.744, 85.877, 0, 21.867, 75.708]
  MoveL 8403 to (-4.56, 58.73, -10.66) mm, rotated rx 180 ry 0 rz 90 deg; joints [75.693, -17.697, 85.758, 0, 21.939, 75.693]
  MoveL 8404 to (-3.08, 58.36, -11.06) mm, rotated rx 180 ry 0 rz 90 deg; joints [75.694, -17.648, 85.633, 0, 22.015, 75.694]
  MoveL 8405 to (-1.56, 58.42, -11.47) mm, rotated rx 180 ry 0 rz 90 deg; joints [75.708, -17.601, 85.513, 0, 22.087, 75.708]
  MoveL 8406 to (-0.12, 58.89, -11.87) mm, rotated rx 180 ry 0 rz 90 deg; joints [75.736, -17.557, 85.406, 0, 22.15, 75.736]
  MoveL 8407 to (1.14, 59.75, -12.28) mm, rotated rx 180 ry 0 rz 90 deg; joints [75.775, -17.517, 85.319, 0, 22.199, 75.775]
  MoveL 8408 to (2.11, 60.91, -12.69) mm, rotated rx -180 ry 0 rz 90 deg; joints [75.821, -17.484, 85.257, 0, 22.228, 75.821]
  MoveL 8409 to (2.73, 62.3, -13.09) mm, rotated rx 180 ry 0 rz 90 deg; joints [75.872, -17.459, 85.224, 0, 22.235, 75.872]
  MoveL 8410 to (2.91, 63.81, -13.5) mm, rotated rx 180 ry 0 rz 90 deg; joints [75.923, -17.441, 85.224, 0, 22.217, 75.923]
  MoveL 8411 to (2.9, 69.03, -13.5) mm, rotated rx -180 ry 0 rz 90 deg; joints [76.095, -17.464, 85.317, 0, 22.148, 76.095]
  MoveC 8412 to (-4.06, 69.3, -13.5) mm, rotated rx -180 ry 0 rz 90 deg; joints [76.047, -17.588, 85.812, 0, 21.776, 76.047] to (-11.02, 69.53, -13.5) mm, rotated rx 180 ry 0 rz 90 deg; joints [75.997, -17.709, 86.305, 0, 21.404, 75.997]
  MoveC 8413 to (-12.97, 67.08, -13.5) mm, rotated rx 180 ry 0 rz 90 deg; joints [75.899, -17.732, 86.399, 0, 21.333, 75.899] to (-12.76, 63.95, -13.5) mm, rotated rx -180 ry 0 rz 90 deg; joints [75.797, -17.715, 86.329, 0, 21.386, 75.797]
  MoveL 8414 to (-5.65, 59.23, -13.5) mm, rotated rx 180 ry 0 rz 90 deg; joints [75.701, -17.572, 85.747, 0, 21.825, 75.701]
  MoveL 8415 to (-4.24, 58.26, -13.5) mm, rotated rx -180 ry 0 rz 90 deg; joints [75.681, -17.543, 85.63, 0, 21.913, 75.681]
  MoveC 8416 to (-4.12, 58.21, -13.5) mm, rotated rx -180 ry 0 rz 90 deg; joints [75.68, -17.54, 85.62, 0, 21.92, 75.68] to (-3.98, 58.2, -13.5) mm, rotated rx -180 ry 0 rz 90 deg; joints [75.681, -17.538, 85.61, 0, 21.927, 75.681]
  MoveC 8417 to (6.42, 59.29, -13.5) mm, rotated rx -180 ry 0 rz 90 deg; joints [75.804, -17.358, 84.894, 0, 22.464, 75.804] to (16.81, 60.53, -13.5) mm, rotated rx 180 ry 0 rz 90 deg; joints [75.93, -17.174, 84.175, 0, 22.999, 75.93]
  MoveL 8418 to (16.81, 68.43, -13.5) mm, rotated rx -180 ry 0 rz 90 deg; joints [76.188, -17.21, 84.315, 0, 22.895, 76.188]
  MoveC 8419 to (9.86, 68.75, -13.5) mm, rotated rx -180 ry 0 rz 90 deg; joints [76.142, -17.338, 84.818, 0, 22.521, 76.142] to (2.9, 69.03, -13.5) mm, rotated rx -180 ry 0 rz 90 deg; joints [76.095, -17.464, 85.317, 0, 22.148, 76.095]
  MoveL 8420 to (2.6, 61.49, -13.5) mm, rotated rx 180 ry 0 rz 90 deg; joints [75.844, -17.436, 85.204, 0, 22.232, 75.844]
  MoveL 8421 to (2.6, 61.49, -10.5) mm, rotated rx -180 ry 0 rz 90 deg; joints [75.844, -17.59, 85.307, 0, 22.284, 75.844]
  Establecer velocidad (1000.0 mm/s)
  MoveL 8422 to (2.6, 61.49, 10) mm, rotated rx 180 ry 0 rz 90 deg; joints [75.844, -18.643, 85.994, 0, 22.649, 75.844]
  Establecer velocidad (66.7 mm/s)
  MoveL 8423 to (14.48, 18.96, 10) mm, rotated rx -180 ry 0 rz 90 deg; joints [74.56, -18.212, 84.349, 0, 23.863, 74.56]
  MoveL 8424 to (14.48, 18.96, -10.25) mm, rotated rx 180 ry 0 rz 90 deg; joints [74.56, -17.179, 83.669, 0, 23.51, 74.56]
  MoveL 8425 to (16.81, 12.74, -12.03) mm, rotated rx -180 ry 0 rz 90 deg; joints [74.38, -17.012, 83.317, 0, 23.695, 74.38]
  MoveL 8426 to (16.81, 18.22, -13.5) mm, rotated rx 180 ry 0 rz 90 deg; joints [74.557, -16.965, 83.376, 0, 23.59, 74.557]
  MoveL 8427 to (16.81, 23.71, -13.5) mm, rotated rx 180 ry 0 rz 90 deg; joints [74.734, -16.994, 83.484, 0, 23.51, 74.734]
  MoveC 8428 to (14.65, 22.67, -13.5) mm, rotated rx 180 ry 0 rz 90 deg; joints [74.681, -17.029, 83.619, 0, 23.41, 74.681] to (13.95, 20.37, -13.5) mm, rotated rx 180 ry 0 rz 90 deg; joints [74.601, -17.03, 83.624, 0, 23.407, 74.601]
  MoveL 8429 to (16.81, 12.74, -13.5) mm, rotated rx -180 ry 0 rz 90 deg; joints [74.38, -16.937, 83.266, 0, 23.67, 74.38]
  MoveL 8430 to (16.81, 18.22, -13.5) mm, rotated rx 180 ry 0 rz 90 deg; joints [74.557, -16.965, 83.376, 0, 23.59, 74.557]
  MoveL 8431 to (16.81, 18.22, -10.5) mm, rotated rx 180 ry 0 rz 90 deg; joints [74.557, -17.119, 83.478, 0, 23.64, 74.557]
  Establecer velocidad (1000.0 mm/s)
  MoveL 8432 to (16.81, 18.22, 10) mm, rotated rx 180 ry 0 rz 90 deg; joints [74.557, -18.163, 84.167, 0, 23.996, 74.557]
  Establecer velocidad (66.7 mm/s)
  MoveL 8433 to (8.58, -67.8, 10) mm, rotated rx -180 ry 0 rz 90 deg; joints [71.738, -17.815, 82.888, 0, 24.927, 71.738]
  MoveL 8434 to (8.58, -67.8, -10.25) mm, rotated rx 180 ry 0 rz 90 deg; joints [71.738, -16.789, 82.207, 0, 24.581, 71.738]
  MoveL 8435 to (10.08, -67.99, -10.66) mm, rotated rx 180 ry 0 rz 90 deg; joints [71.748, -16.737, 82.081, 0, 24.656, 71.748]
  MoveL 8436 to (11.59, -67.8, -11.06) mm, rotated rx 180 ry 0 rz 90 deg; joints [71.769, -16.688, 81.963, 0, 24.725, 71.769]
  MoveL 8437 to (13.02, -67.29, -11.47) mm, rotated rx -180 ry 0 rz 90 deg; joints [71.8, -16.643, 81.858, 0, 24.785, 71.8]
  MoveL 8438 to (14.3, -66.47, -11.87) mm, rotated rx -180 ry 0 rz 90 deg; joints [71.839, -16.602, 81.771, 0, 24.831, 71.839]
  MoveL 8439 to (15.37, -65.39, -12.28) mm, rotated rx -180 ry 0 rz 90 deg; joints [71.883, -16.567, 81.705, 0, 24.862, 71.883]
  MoveL 8440 to (16.18, -64.11, -12.69) mm, rotated rx 180 ry 0 rz 90 deg; joints [71.932, -16.539, 81.664, 0, 24.875, 71.932]
  MoveL 8441 to (16.68, -62.67, -13.09) mm, rotated rx -180 ry 0 rz 90 deg; joints [71.982, -16.518, 81.648, 0, 24.87, 71.982]
  MoveL 8442 to (16.81, -61.16, -13.5) mm, rotated rx -180 ry 0 rz 90 deg; joints [72.031, -16.504, 81.659, 0, 24.845, 72.031]
  MoveL 8443 to (16.81, -52.45, -13.5) mm, rotated rx -180 ry 0 rz 90 deg; joints [72.305, -16.56, 81.861, 0, 24.698, 72.305]
  MoveL 8444 to (16.81, -36.3, -13.5) mm, rotated rx 180 ry 0 rz 90 deg; joints [72.815, -16.659, 82.227, 0, 24.432, 72.815]
  MoveL 8445 to (14.69, -34.5, -13.5) mm, rotated rx -180 ry 0 rz 90 deg; joints [72.851, -16.711, 82.421, 0, 24.291, 72.851]
  MoveL 8446 to (14.5, -34.35, -13.5) mm, rotated rx -180 ry 0 rz 90 deg; joints [72.854, -16.716, 82.438, 0, 24.278, 72.854]
  MoveC 8447 to (12.57, -33.95, -13.5) mm, rotated rx -180 ry 0 rz 90 deg; joints [72.848, -16.755, 82.585, 0, 24.17, 72.848] to (10.71, -34.61, -13.5) mm, rotated rx -180 ry 0 rz 90 deg; joints [72.809, -16.787, 82.704, 0, 24.083, 72.809]
  MoveC 8448 to (10.26, -35.06, -13.5) mm, rotated rx 180 ry 0 rz 90 deg; joints [72.79, -16.793, 82.726, 0, 24.067, 72.79] to (9.99, -35.64, -13.5) mm, rotated rx 180 ry 0 rz 90 deg; joints [72.769, -16.795, 82.732, 0, 24.062, 72.769]
  MoveL 8449 to (1.94, -64.91, -13.5) mm, rotated rx -180 ry 0 rz 90 deg; joints [71.76, -16.77, 82.639, 0, 24.131, 71.76]
  MoveL 8450 to (1.69, -65.88, -13.5) mm, rotated rx -180 ry 0 rz 90 deg; joints [71.727, -16.768, 82.634, 0, 24.135, 71.727]
  MoveC 8451 to (1.64, -66.67, -13.5) mm, rotated rx -180 ry 0 rz 90 deg; joints [71.701, -16.764, 82.619, 0, 24.146, 71.701] to (1.89, -67.42, -13.5) mm, rotated rx -180 ry 0 rz 90 deg; joints [71.68, -16.755, 82.583, 0, 24.172, 71.68]
  MoveL 8452 to (2.03, -67.66, -13.5) mm, rotated rx -180 ry 0 rz 90 deg; joints [71.674, -16.751, 82.568, 0, 24.183, 71.674]
  MoveC 8453 to (3.13, -68.77, -13.5) mm, rotated rx -180 ry 0 rz 90 deg; joints [71.65, -16.722, 82.462, 0, 24.26, 71.65] to (4.66, -69.15, -13.5) mm, rotated rx -180 ry 0 rz 90 deg; joints [71.655, -16.691, 82.345, 0, 24.346, 71.655]
  MoveL 8454 to (5.21, -69.13, -13.5) mm, rotated rx -180 ry 0 rz 90 deg; joints [71.661, -16.68, 82.305, 0, 24.375, 71.661]
  MoveL 8455 to (15.64, -68.67, -13.5) mm, rotated rx 180 ry 0 rz 90 deg; joints [71.783, -16.479, 81.567, 0, 24.912, 71.783]
  MoveL 8456 to (16.81, -68.6, -13.5) mm, rotated rx 180 ry 0 rz 90 deg; joints [71.798, -16.456, 81.483, 0, 24.973, 71.798]
  MoveL 8457 to (16.81, -52.45, -13.5) mm, rotated rx -180 ry 0 rz 90 deg; joints [72.305, -16.56, 81.861, 0, 24.698, 72.305]
  MoveL 8458 to (9.27, -52.45, -13.5) mm, rotated rx 180 ry 0 rz 90 deg; joints [72.229, -16.707, 82.404, 0, 24.302, 72.229]
  MoveL 8459 to (9.27, -52.45, -10.5) mm, rotated rx 180 ry 0 rz 90 deg; joints [72.229, -16.859, 82.507, 0, 24.352, 72.229]
  Establecer velocidad (1000.0 mm/s)
  MoveL 8460 to (9.27, -52.45, 10) mm, rotated rx -180 ry 0 rz 90 deg; joints [72.229, -17.9, 83.197, 0, 24.704, 72.229]
  Establecer velocidad (66.7 mm/s)
  MoveL 8461 to (-39.19, -52.09, 10) mm, rotated rx -180 ry 0 rz 90 deg; joints [71.736, -18.799, 86.608, 0, 22.191, 71.736]
  MoveL 8462 to (-39.19, -52.09, -10.25) mm, rotated rx 180 ry 0 rz 90 deg; joints [71.736, -17.757, 85.929, 0, 21.828, 71.736]
  MoveL 8463 to (-37.78, -52.64, -10.66) mm, rotated rx 180 ry 0 rz 90 deg; joints [71.733, -17.709, 85.805, 0, 21.903, 71.733]
  MoveL 8464 to (-36.27, -52.84, -11.06) mm, rotated rx 180 ry 0 rz 90 deg; joints [71.743, -17.661, 85.683, 0, 21.978, 71.743]
  MoveL 8465 to (-34.75, -52.7, -11.47) mm, rotated rx 180 ry 0 rz 90 deg; joints [71.764, -17.614, 85.567, 0, 22.047, 71.764]
  MoveL 8466 to (-33.31, -52.23, -11.87) mm, rotated rx 180 ry 0 rz 90 deg; joints [71.794, -17.571, 85.464, 0, 22.107, 71.794]
